LIN {X 0,Y 418.203,Z 303.395,A -85,B 0,C 180,E1 -10039.132,E2 -10039.132} C_VEL
LIN {X 0,Y 418.231,Z 303.386,A -85,B 0,C 180,E1 -10042.775,E2 -10042.775} C_VEL
LIN {X 0,Y 418.224,Z 303.373,A -85,B 0,C 180,E1 -10046.321,E2 -10046.321} C_VEL
LIN {X 0,Y 418.233,Z 303.387,A -85,B 0,C 180,E1 -10049.727,E2 -10049.727} C_VEL
LIN {X 0,Y 418.217,Z 303.388,A -85,B 0,C 180,E1 -10053.017,E2 -10053.017} C_VEL
LIN {X 0,Y 418.247,Z 303.384,A -85,B 0,C 180,E1 -10056.217,E2 -10056.217} C_VEL
LIN {X 0,Y 418.24,Z 303.384,A -85,B 0,C 180,E1 -10059.337,E2 -10059.337} C_VEL
LIN {X 0,Y 418.246,Z 303.382,A -85,B 0,C 180,E1 -10062.395,E2 -10062.395} C_VEL
LIN {X 0,Y 418.265,Z 303.381,A -85,B 0,C 180,E1 -10065.402,E2 -10065.402} C_VEL
LIN {X 0,Y 418.292,Z 303.381,A -85,B 0,C 180,E1 -10068.369,E2 -10068.369} C_VEL
LIN {X 0,Y 418.437,Z 303.357,A -85,B 0,C 180,E1 -10072.278,E2 -10072.278} C_VEL
LIN {X 0,Y 418.453,Z 303.363,A -85,B 0,C 180,E1 -10074.217,E2 -10074.217} C_VEL
LIN {X 0,Y 418.521,Z 303.346,A -85,B 0,C 180,E1 -10078.076,E2 -10078.076} C_VEL
LIN {X 0,Y 418.461,Z 303.353,A -85,B 0,C 180,E1 -10080.963,E2 -10080.963} C_VEL
LIN {X 0,Y 418.457,Z 303.356,A -85,B 0,C 180,E1 -10082.888,E2 -10082.888} C_VEL
LIN {X 0,Y 418.488,Z 303.352,A -85,B 0,C 180,E1 -10085.783,E2 -10085.783} C_VEL
LIN {X 0,Y 418.36,Z 303.365,A -85,B 0,C 180,E1 -10088.696,E2 -10088.696} C_VEL
LIN {X 0,Y 418.302,Z 303.372,A -85,B 0,C 180,E1 -10091.632,E2 -10091.632} C_VEL
LIN {X 0,Y 418.289,Z 303.374,A -85,B 0,C 180,E1 -10094.598,E2 -10094.598} C_VEL
LIN {X 0,Y 418.27,Z 303.372,A -85,B 0,C 180,E1 -10097.605,E2 -10097.605} C_VEL
LIN {X 0,Y 418.242,Z 303.384,A -85,B 0,C 180,E1 -10100.664,E2 -10100.664} C_VEL
LIN {X 0,Y 418.251,Z 303.38,A -85,B 0,C 180,E1 -10103.784,E2 -10103.784} C_VEL
LIN {X 0,Y 418.217,Z 303.387,A -85,B 0,C 180,E1 -10107.048,E2 -10107.048} C_VEL
LIN {X 0,Y 418.235,Z 303.384,A -85,B 0,C 180,E1 -10110.273,E2 -10110.273} C_VEL
LIN {X 0,Y 418.242,Z 303.388,A -85,B 0,C 180,E1 -10113.678,E2 -10113.678} C_VEL
LIN {X 0,Y 418.232,Z 303.388,A -85,B 0,C 180,E1 -10117.225,E2 -10117.225} C_VEL
LIN {X 0,Y 418.207,Z 303.39,A -85,B 0,C 180,E1 -10120.869,E2 -10120.869} C_VEL
LIN {X 0,Y 418.203,Z 303.38,A -85,B 0,C 180,E1 -10123.73,E2 -10123.73} C_VEL
LIN {X 0,Y 418.203,Z 303.392,A -85,B 0,C 180,E1 -10126.449,E2 -10126.449} C_VEL
LIN {X 0,Y 418.217,Z 303.391,A -85,B 0,C 180,E1 -10129.132,E2 -10129.132} C_VEL
LIN {X 0,Y 418.221,Z 303.393,A -85,B 0,C 180,E1 -10132.168,E2 -10132.168} C_VEL
LIN {X 0,Y 418.262,Z 303.379,A -85,B 0,C 180,E1 -10135.421,E2 -10135.421} C_VEL
LIN {X 0,Y 418.21,Z 303.393,A -85,B 0,C 180,E1 -10138.605,E2 -10138.605} C_VEL
LIN {X 0,Y 418.318,Z 303.393,A -85,B 0,C 180,E1 -10142.251,E2 -10142.251} C_VEL
LIN {X 0,Y 420.764,Z 315.163,A -85,B 0,C 180,E1 -10144.934,E2 -10144.934} C_VEL
LIN {X 0,Y 421.568,Z 320.765,A -85,B 0,C 180,E1 -10146.155,E2 -10146.155} C_VEL
LIN {X 0,Y 420.324,Z 337.886,A -85,B 0,C 180,E1 -10149.597,E2 -10149.597} C_VEL
LIN {X 0,Y 420,Z 342.885,A -85,B 0,C 180,E1 -10150.591,E2 -10150.591} C_VEL
LIN {X 0,Y 423.729,Z 363.444,A -85,B 0,C 180,E1 -10151.164,E2 -10151.164} C_VEL
LIN {X 0,Y 424.474,Z 370.034,A -85,B 0,C 180,E1 -10151.321,E2 -10151.321} C_VEL
LIN {X 0,Y 423.504,Z 451.222,A -85,B 0,C 180,E1 -10152.746,E2 -10152.746} C_VEL
LIN {X 0,Y 422.93,Z 464.392,A -85,B 0,C 180,E1 -10153.157,E2 -10153.157} C_VEL
LIN {X 0,Y 422.257,Z 477.049,A -85,B 0,C 180,E1 -10153.751,E2 -10153.751} C_VEL
LIN {X 0,Y 421.448,Z 489.124,A -85,B 0,C 180,E1 -10154.526,E2 -10154.526} C_VEL
LIN {X 0,Y 420.581,Z 500.615,A -85,B 0,C 180,E1 -10155.485,E2 -10155.485} C_VEL
LIN {X 0,Y 419.836,Z 510.983,A -85,B 0,C 180,E1 -10156.571,E2 -10156.571} C_VEL
LIN {X 0,Y 419.198,Z 519.483,A -85,B 0,C 180,E1 -10157.658,E2 -10157.658} C_VEL
LIN {X 0,Y 418.464,Z 527.341,A -85,B 0,C 180,E1 -10158.865,E2 -10158.865} C_VEL
LIN {X 0,Y 417.91,Z 535.031,A -85,B 0,C 180,E1 -10160.32,E2 -10160.32} C_VEL
LIN {X 0,Y 417.502,Z 541.222,A -85,B 0,C 180,E1 -10161.775,E2 -10161.775} C_VEL
LIN {X 0,Y 417.242,Z 546.152,A -85,B 0,C 180,E1 -10163.23,E2 -10163.23} C_VEL
LIN {X 0,Y 417.122,Z 549.965,A -85,B 0,C 180,E1 -10164.684,E2 -10164.684} C_VEL
LIN {X 0,Y 417.013,Z 552.763,A -85,B 0,C 180,E1 -10166.136,E2 -10166.136} C_VEL
LIN {X 0,Y 417.056,Z 555.025,A -85,B 0,C 180,E1 -10168.069,E2 -10168.069} C_VEL
LIN {X 0,Y 417.011,Z 555.562,A -85,B 0,C 180,E1 -10169.035,E2 -10169.035} C_VEL
LIN {X 0,Y 417.004,Z 555.667,A -85,B 0,C 180,E1 -10170.001,E2 -10170.001} C_VEL
LIN {X 0,Y 417.056,Z 554.713,A -85,B 0,C 180,E1 -10171.932,E2 -10171.932} C_VEL
LIN {X 0,Y 417.03,Z 553.643,A -85,B 0,C 180,E1 -10172.899,E2 -10172.899} C_VEL
LIN {X 0,Y 417.015,Z 552.117,A -85,B 0,C 180,E1 -10173.866,E2 -10173.866} C_VEL
LIN {X 0,Y 417.122,Z 549.039,A -85,B 0,C 180,E1 -10175.318,E2 -10175.318} C_VEL
LIN {X 0,Y 417.233,Z 544.889,A -85,B 0,C 180,E1 -10176.772,E2 -10176.772} C_VEL
LIN {X 0,Y 417.504,Z 538.537,A -85,B 0,C 180,E1 -10178.471,E2 -10178.471} C_VEL
LIN {X 0,Y 417.901,Z 531.613,A -85,B 0,C 180,E1 -10179.927,E2 -10179.927} C_VEL
LIN {X 0,Y 418.308,Z 524.531,A -85,B 0,C 180,E1 -10181.141,E2 -10181.141} C_VEL
LIN {X 0,Y 418.943,Z 515.991,A -85,B 0,C 180,E1 -10182.351,E2 -10182.351} C_VEL
LIN {X 0,Y 419.634,Z 505.417,A -85,B 0,C 180,E1 -10183.561,E2 -10183.561} C_VEL
LIN {X 0,Y 420.269,Z 494.939,A -85,B 0,C 180,E1 -10184.528,E2 -10184.528} C_VEL
LIN {X 0,Y 420.952,Z 483.424,A -85,B 0,C 180,E1 -10185.37,E2 -10185.37} C_VEL
LIN {X 0,Y 421.546,Z 471.495,A -85,B 0,C 180,E1 -10186.03,E2 -10186.03} C_VEL
LIN {X 0,Y 422.09,Z 458.63,A -85,B 0,C 180,E1 -10186.537,E2 -10186.537} C_VEL
LIN {X 0,Y 422.434,Z 445.189,A -85,B 0,C 180,E1 -10186.865,E2 -10186.865} C_VEL
LIN {X 0,Y 423.121,Z 367.493,A -85,B 0,C 180,E1 -10188.19,E2 -10188.19} C_VEL
LIN {X 0,Y 419.458,Z 343.088,A -85,B 0,C 180,E1 -10188.785,E2 -10188.785} C_VEL
LIN {X 0,Y 420.548,Z 324.975,A -85,B 0,C 180,E1 -10192.346,E2 -10192.346} C_VEL
LIN {X 0,Y 420.862,Z 317.24,A -85,B 0,C 180,E1 -10193.889,E2 -10193.889} C_VEL
LIN {X 0,Y 418.323,Z 303.378,A -85,B 0,C 180,E1 -10196.875,E2 -10196.875} C_VEL
LIN {X 0,Y 418.249,Z 303.384,A -85,B 0,C 180,E1 -10200.272,E2 -10200.272} C_VEL
LIN {X 0,Y 418.253,Z 303.385,A -85,B 0,C 180,E1 -10203.677,E2 -10203.677} C_VEL
LIN {X 0,Y 418.242,Z 303.382,A -85,B 0,C 180,E1 -10207.225,E2 -10207.225} C_VEL
LIN {X 0,Y 418.213,Z 303.387,A -85,B 0,C 180,E1 -10210.868,E2 -10210.868} C_VEL
LIN {X 0,Y 418.212,Z 303.387,A -85,B 0,C 180,E1 -10213.729,E2 -10213.729} C_VEL
LIN {X 0,Y 418.212,Z 303.394,A -85,B 0,C 180,E1 -10216.449,E2 -10216.449} C_VEL
LIN {X 0,Y 418.225,Z 303.385,A -85,B 0,C 180,E1 -10219.131,E2 -10219.131} C_VEL
LIN {X 0,Y 418.228,Z 303.386,A -85,B 0,C 180,E1 -10222.168,E2 -10222.168} C_VEL
LIN {X 0,Y 418.269,Z 303.38,A -85,B 0,C 180,E1 -10225.42,E2 -10225.42} C_VEL
LIN {X 0,Y 418.215,Z 303.389,A -85,B 0,C 180,E1 -10228.604,E2 -10228.604} C_VEL
LIN {X 0,Y 418.265,Z 303.379,A -85,B 0,C 180,E1 -10231.934,E2 -10231.934} C_VEL
LIN {X 0,Y 418.276,Z 303.386,A -85,B 0,C 180,E1 -10235.162,E2 -10235.162} C_VEL
LIN {X 0,Y 418.238,Z 303.382,A -85,B 0,C 180,E1 -10238.304,E2 -10238.304} C_VEL
LIN {X 0,Y 418.281,Z 303.385,A -85,B 0,C 180,E1 -10241.383,E2 -10241.383} C_VEL
LIN {X 0,Y 418.305,Z 303.374,A -85,B 0,C 180,E1 -10244.406,E2 -10244.406} C_VEL
LIN {X 0,Y 418.359,Z 303.372,A -85,B 0,C 180,E1 -10247.385,E2 -10247.385} C_VEL
LIN {X 0,Y 418.34,Z 303.371,A -85,B 0,C 180,E1 -10250.328,E2 -10250.328} C_VEL
LIN {X 0,Y 418.471,Z 303.355,A -85,B 0,C 180,E1 -10253.248,E2 -10253.248} C_VEL
LIN {X 0,Y 418.331,Z 303.371,A -85,B 0,C 180,E1 -10255.181,E2 -10255.181} C_VEL
LIN {X 0,Y 418.542,Z 303.352,A -85,B 0,C 180,E1 -10258.075,E2 -10258.075} C_VEL
LIN {X 0,Y 418.67,Z 303.335,A -85,B 0,C 180,E1 -10260,E2 -10260} C_VEL
LIN {X 0,Y 418.494,Z 303.351,A -85,B 0,C 180,E1 -10262.888,E2 -10262.888} C_VEL
LIN {X 0,Y 418.447,Z 303.358,A -85,B 0,C 180,E1 -10266.548,E2 -10266.548} C_VEL
LIN {X 0,Y 418.342,Z 303.37,A -85,B 0,C 180,E1 -10269.671,E2 -10269.671} C_VEL
LIN {X 0,Y 418.35,Z 303.372,A -85,B 0,C 180,E1 -10273,E2 -10273} C_VEL
LIN {X 0,Y 418.316,Z 303.381,A -85,B 0,C 180,E1 -10276.735,E2 -10276.735} C_VEL
LIN {X 0,Y 418.273,Z 303.378,A -85,B 0,C 180,E1 -10279.79,E2 -10279.79} C_VEL
LIN {X 0,Y 418.234,Z 303.388,A -85,B 0,C 180,E1 -10282.736,E2 -10282.736} C_VEL
LIN {X 0,Y 418.24,Z 303.383,A -85,B 0,C 180,E1 -10285.906,E2 -10285.906} C_VEL
LIN {X 0,Y 418.263,Z 303.387,A -85,B 0,C 180,E1 -10289.162,E2 -10289.162} C_VEL
LIN {X 0,Y 418.259,Z 303.382,A -85,B 0,C 180,E1 -10292.843,E2 -10292.843} C_VEL
LIN {X 0,Y 418.245,Z 303.382,A -85,B 0,C 180,E1 -10296.237,E2 -10296.237} C_VEL
LIN {X 0,Y 418.244,Z 303.389,A -85,B 0,C 180,E1 -10299.683,E2 -10299.683} C_VEL
LIN {X 0,Y 418.225,Z 303.385,A -85,B 0,C 180,E1 -10302.32,E2 -10302.32} C_VEL
LIN {X 0,Y 418.237,Z 303.383,A -85,B 0,C 180,E1 -10305.108,E2 -10305.108} C_VEL
LIN {X 0,Y 418.236,Z 303.389,A -85,B 0,C 180,E1 -10307.765,E2 -10307.765} C_VEL
LIN {X 0,Y 418.244,Z 303.384,A -85,B 0,C 180,E1 -10311.556,E2 -10311.556} C_VEL
LIN {X 0,Y 418.26,Z 303.38,A -85,B 0,C 180,E1 -10315.158,E2 -10315.158} C_VEL
LIN {X 0,Y 418.247,Z 303.381,A -85,B 0,C 180,E1 -10317.471,E2 -10317.471} C_VEL
LIN {X 0,Y 418.266,Z 303.382,A -85,B 0,C 180,E1 -10320.896,E2 -10320.896} C_VEL
LIN {X 0,Y 418.238,Z 303.385,A -85,B 0,C 180,E1 -10324.093,E2 -10324.093} C_VEL
LIN {X 0,Y 418.238,Z 303.384,A -85,B 0,C 180,E1 -10327.263,E2 -10327.263} C_VEL
LIN {X 0,Y 418.284,Z 303.379,A -85,B 0,C 180,E1 -10330.363,E2 -10330.363} C_VEL
LIN {X 0,Y 418.317,Z 303.375,A -85,B 0,C 180,E1 -10333.404,E2 -10333.404} C_VEL
LIN {X 0,Y 418.347,Z 303.376,A -85,B 0,C 180,E1 -10336.999,E2 -10336.999} C_VEL
LIN {X 0,Y 418.357,Z 303.373,A -85,B 0,C 180,E1 -10340.816,E2 -10340.816} C_VEL
LIN {X 0,Y 418.382,Z 303.531,A -85,B 0,C 180,E1 -10341.304,E2 -10341.304} C_VEL
LIN {X 0,Y 419.874,Z 311.987,A -85,B 0,C 180,E1 -10343.27,E2 -10343.27} C_VEL
LIN {X 0,Y 419.639,Z 321.318,A -85,B 0,C 180,E1 -10345.314,E2 -10345.314} C_VEL
LIN {X 0,Y 423.403,Z 342.206,A -85,B 0,C 180,E1 -10345.831,E2 -10345.831} C_VEL
LIN {X 0,Y 422.409,Z 428.625,A -85,B 0,C 180,E1 -10347.32,E2 -10347.32} C_VEL
LIN {X 0,Y 422.171,Z 435.313,A -85,B 0,C 180,E1 -10347.505,E2 -10347.505} C_VEL
LIN {X 0,Y 420.767,Z 442.88,A -85,B 0,C 180,E1 -10347.736,E2 -10347.736} C_VEL
LIN {X 0,Y 418.093,Z 450.166,A -85,B 0,C 180,E1 -10347.981,E2 -10347.981} C_VEL
LIN {X 0,Y 415.016,Z 459.136,A -85,B 0,C 180,E1 -10348.398,E2 -10348.398} C_VEL
LIN {X 0,Y 414.153,Z 464.405,A -85,B 0,C 180,E1 -10348.731,E2 -10348.731} C_VEL
LIN {X 0,Y 413.477,Z 475.677,A -85,B 0,C 180,E1 -10349.634,E2 -10349.634} C_VEL
LIN {X 0,Y 412.722,Z 486.46,A -85,B 0,C 180,E1 -10350.731,E2 -10350.731} C_VEL
LIN {X 0,Y 412.056,Z 496.153,A -85,B 0,C 180,E1 -10351.954,E2 -10351.954} C_VEL
LIN {X 0,Y 411.442,Z 504.117,A -85,B 0,C 180,E1 -10353.181,E2 -10353.181} C_VEL
LIN {X 0,Y 410.924,Z 511.91,A -85,B 0,C 180,E1 -10354.659,E2 -10354.659} C_VEL
LIN {X 0,Y 410.603,Z 518.384,A -85,B 0,C 180,E1 -10356.208,E2 -10356.208} C_VEL
LIN {X 0,Y 410.256,Z 523.824,A -85,B 0,C 180,E1 -10357.876,E2 -10357.876} C_VEL
LIN {X 0,Y 410.051,Z 527.487,A -85,B 0,C 180,E1 -10359.37,E2 -10359.37} C_VEL
LIN {X 0,Y 409.963,Z 530.119,A -85,B 0,C 180,E1 -10360.869,E2 -10360.869} C_VEL
LIN {X 0,Y 409.905,Z 531.676,A -85,B 0,C 180,E1 -10362.235,E2 -10362.235} C_VEL
LIN {X 0,Y 409.789,Z 532.527,A -85,B 0,C 180,E1 -10363.892,E2 -10363.892} C_VEL
LIN {X 0,Y 409.806,Z 532.503,A -85,B 0,C 180,E1 -10364.906,E2 -10364.906} C_VEL
LIN {X 0,Y 409.886,Z 531.827,A -85,B 0,C 180,E1 -10366.222,E2 -10366.222} C_VEL
LIN {X 0,Y 409.974,Z 529.837,A -85,B 0,C 180,E1 -10367.972,E2 -10367.972} C_VEL
LIN {X 0,Y 410.241,Z 526.867,A -85,B 0,C 180,E1 -10369.572,E2 -10369.572} C_VEL
LIN {X 0,Y 410.504,Z 523.013,A -85,B 0,C 180,E1 -10371.07,E2 -10371.07} C_VEL
LIN {X 0,Y 410.967,Z 517.198,A -85,B 0,C 180,E1 -10372.785,E2 -10372.785} C_VEL
LIN {X 0,Y 411.614,Z 509.788,A -85,B 0,C 180,E1 -10374.458,E2 -10374.458} C_VEL
LIN {X 0,Y 412.182,Z 502.894,A -85,B 0,C 180,E1 -10375.717,E2 -10375.717} C_VEL
LIN {X 0,Y 412.992,Z 493.798,A -85,B 0,C 180,E1 -10377.077,E2 -10377.077} C_VEL
LIN {X 0,Y 413.829,Z 484.223,A -85,B 0,C 180,E1 -10378.232,E2 -10378.232} C_VEL
LIN {X 0,Y 414.719,Z 473.231,A -85,B 0,C 180,E1 -10379.295,E2 -10379.295} C_VEL
LIN {X 0,Y 415.533,Z 461.267,A -85,B 0,C 180,E1 -10380.209,E2 -10380.209} C_VEL
LIN {X 0,Y 416.24,Z 448.697,A -85,B 0,C 180,E1 -10380.924,E2 -10380.924} C_VEL
LIN {X 0,Y 416.732,Z 435.712,A -85,B 0,C 180,E1 -10381.448,E2 -10381.448} C_VEL
LIN {X 0,Y 417.033,Z 422.429,A -85,B 0,C 180,E1 -10381.777,E2 -10381.777} C_VEL
LIN {X 0,Y 418.216,Z 343.018,A -85,B 0,C 180,E1 -10383.163,E2 -10383.163} C_VEL
LIN {X 0,Y 413.927,Z 323.175,A -85,B 0,C 180,E1 -10383.775,E2 -10383.775} C_VEL
LIN {X 0,Y 413.523,Z 321.336,A -85,B 0,C 180,E1 -10383.87,E2 -10383.87} C_VEL
LIN {X 0,Y 413.629,Z 316.261,A -85,B 0,C 180,E1 -10384.99,E2 -10384.99} C_VEL
LIN {X 0,Y 411.392,Z 305.21,A -85,B 0,C 180,E1 -10387.641,E2 -10387.641} C_VEL
LIN {X 0,Y 411.195,Z 304.267,A -85,B 0,C 180,E1 -10387.894,E2 -10387.894} C_VEL
LIN {X 0,Y 411.145,Z 304.269,A -85,B 0,C 180,E1 -10391.226,E2 -10391.226} C_VEL
LIN {X 0,Y 411.168,Z 304.269,A -85,B 0,C 180,E1 -10394.49,E2 -10394.49} C_VEL
LIN {X 0,Y 411.156,Z 304.266,A -85,B 0,C 180,E1 -10398.192,E2 -10398.192} C_VEL
LIN {X 0,Y 411.188,Z 304.263,A -85,B 0,C 180,E1 -10401.832,E2 -10401.832} C_VEL
LIN {X 0,Y 411.195,Z 304.258,A -85,B 0,C 180,E1 -10405.123,E2 -10405.123} C_VEL
LIN {X 0,Y 411.155,Z 304.269,A -85,B 0,C 180,E1 -10408.002,E2 -10408.002} C_VEL
LIN {X 0,Y 411.184,Z 304.264,A -85,B 0,C 180,E1 -10411.408,E2 -10411.408} C_VEL
LIN {X 0,Y 411.203,Z 304.258,A -85,B 0,C 180,E1 -10414.934,E2 -10414.934} C_VEL
LIN {X 0,Y 411.194,Z 304.261,A -85,B 0,C 180,E1 -10417.913,E2 -10417.913} C_VEL
LIN {X 0,Y 411.205,Z 304.259,A -85,B 0,C 180,E1 -10421.051,E2 -10421.051} C_VEL
LIN {X 0,Y 411.199,Z 304.265,A -85,B 0,C 180,E1 -10424.13,E2 -10424.13} C_VEL
LIN {X 0,Y 411.292,Z 304.242,A -85,B 0,C 180,E1 -10427.166,E2 -10427.166} C_VEL
LIN {X 0,Y 411.264,Z 304.253,A -85,B 0,C 180,E1 -10430.161,E2 -10430.161} C_VEL
LIN {X 0,Y 411.375,Z 304.237,A -85,B 0,C 180,E1 -10433.132,E2 -10433.132} C_VEL
LIN {X 0,Y 411.271,Z 304.249,A -85,B 0,C 180,E1 -10435.099,E2 -10435.099} C_VEL
LIN {X 0,Y 411.49,Z 304.222,A -85,B 0,C 180,E1 -10438.043,E2 -10438.043} C_VEL
LIN {X 0,Y 411.426,Z 304.229,A -85,B 0,C 180,E1 -10440.979,E2 -10440.979} C_VEL
LIN {X 0,Y 411.415,Z 304.233,A -85,B 0,C 180,E1 -10442.938,E2 -10442.938} C_VEL
LIN {X 0,Y 411.422,Z 304.228,A -85,B 0,C 180,E1 -10446.868,E2 -10446.868} C_VEL
LIN {X 0,Y 411.273,Z 304.249,A -85,B 0,C 180,E1 -10449.839,E2 -10449.839} C_VEL
LIN {X 0,Y 411.297,Z 304.243,A -85,B 0,C 180,E1 -10453.104,E2 -10453.104} C_VEL
LIN {X 0,Y 411.249,Z 304.255,A -85,B 0,C 180,E1 -10456.889,E2 -10456.889} C_VEL
LIN {X 0,Y 411.223,Z 304.255,A -85,B 0,C 180,E1 -10459.987,E2 -10459.987} C_VEL
LIN {X 0,Y 411.181,Z 304.26,A -85,B 0,C 180,E1 -10463.149,E2 -10463.149} C_VEL
LIN {X 0,Y 411.177,Z 304.262,A -85,B 0,C 180,E1 -10466.385,E2 -10466.385} C_VEL
LIN {X 0,Y 411.191,Z 304.265,A -85,B 0,C 180,E1 -10469.714,E2 -10469.714} C_VEL
LIN {X 0,Y 411.2,Z 304.263,A -85,B 0,C 180,E1 -10473.157,E2 -10473.157} C_VEL
LIN {X 0,Y 411.186,Z 304.262,A -85,B 0,C 180,E1 -10476.553,E2 -10476.553} C_VEL
LIN {X 0,Y 411.171,Z 304.268,A -85,B 0,C 180,E1 -10479.723,E2 -10479.723} C_VEL
LIN {X 0,Y 411.165,Z 304.256,A -85,B 0,C 180,E1 -10483.135,E2 -10483.135} C_VEL
LIN {X 0,Y 411.163,Z 304.274,A -85,B 0,C 180,E1 -10485.882,E2 -10485.882} C_VEL
LIN {X 0,Y 411.156,Z 304.27,A -85,B 0,C 180,E1 -10488.773,E2 -10488.773} C_VEL
LIN {X 0,Y 411.186,Z 304.269,A -85,B 0,C 180,E1 -10492.027,E2 -10492.027} C_VEL
LIN {X 0,Y 411.203,Z 304.259,A -85,B 0,C 180,E1 -10495.668,E2 -10495.668} C_VEL
LIN {X 0,Y 411.187,Z 304.267,A -85,B 0,C 180,E1 -10499.154,E2 -10499.154} C_VEL
LIN {X 0,Y 411.265,Z 304.258,A -85,B 0,C 180,E1 -10501.902,E2 -10501.902} C_VEL
LIN {X 0,Y 413.59,Z 315.249,A -85,B 0,C 180,E1 -10504.471,E2 -10504.471} C_VEL
LIN {X 0,Y 414.671,Z 322.091,A -85,B 0,C 180,E1 -10506,E2 -10506} C_VEL
LIN {X 0,Y 413.41,Z 338.62,A -85,B 0,C 180,E1 -10509.38,E2 -10509.38} C_VEL
LIN {X 0,Y 413.181,Z 342.913,A -85,B 0,C 180,E1 -10510.208,E2 -10510.208} C_VEL
LIN {X 0,Y 417.065,Z 363.859,A -85,B 0,C 180,E1 -10510.814,E2 -10510.814} C_VEL
LIN {X 0,Y 417.867,Z 370.718,A -85,B 0,C 180,E1 -10510.983,E2 -10510.983} C_VEL
LIN {X 0,Y 416.829,Z 451.568,A -85,B 0,C 180,E1 -10512.429,E2 -10512.429} C_VEL
LIN {X 0,Y 416.203,Z 464.561,A -85,B 0,C 180,E1 -10512.845,E2 -10512.845} C_VEL
LIN {X 0,Y 415.484,Z 477.666,A -85,B 0,C 180,E1 -10513.479,E2 -10513.479} C_VEL
LIN {X 0,Y 414.636,Z 489.507,A -85,B 0,C 180,E1 -10514.266,E2 -10514.266} C_VEL
LIN {X 0,Y 413.735,Z 500.891,A -85,B 0,C 180,E1 -10515.239,E2 -10515.239} C_VEL
LIN {X 0,Y 412.922,Z 511.174,A -85,B 0,C 180,E1 -10516.341,E2 -10516.341} C_VEL
LIN {X 0,Y 412.25,Z 519.598,A -85,B 0,C 180,E1 -10517.447,E2 -10517.447} C_VEL
LIN {X 0,Y 411.368,Z 528.752,A -85,B 0,C 180,E1 -10518.92,E2 -10518.92} C_VEL
LIN {X 0,Y 410.8,Z 536.134,A -85,B 0,C 180,E1 -10520.399,E2 -10520.399} C_VEL
LIN {X 0,Y 410.345,Z 542.951,A -85,B 0,C 180,E1 -10522.126,E2 -10522.126} C_VEL
LIN {X 0,Y 410.043,Z 547.898,A -85,B 0,C 180,E1 -10523.776,E2 -10523.776} C_VEL
LIN {X 0,Y 410.019,Z 550.906,A -85,B 0,C 180,E1 -10525.084,E2 -10525.084} C_VEL
LIN {X 0,Y 409.924,Z 553.935,A -85,B 0,C 180,E1 -10527.053,E2 -10527.053} C_VEL
LIN {X 0,Y 409.966,Z 554.858,A -85,B 0,C 180,E1 -10528.036,E2 -10528.036} C_VEL
LIN {X 0,Y 409.935,Z 555.373,A -85,B 0,C 180,E1 -10529.019,E2 -10529.019} C_VEL
LIN {X 0,Y 409.936,Z 555.165,A -85,B 0,C 180,E1 -10530.983,E2 -10530.983} C_VEL
LIN {X 0,Y 409.967,Z 554.482,A -85,B 0,C 180,E1 -10531.966,E2 -10531.966} C_VEL
LIN {X 0,Y 409.929,Z 553.39,A -85,B 0,C 180,E1 -10532.949,E2 -10532.949} C_VEL
LIN {X 0,Y 409.933,Z 551.846,A -85,B 0,C 180,E1 -10533.933,E2 -10533.933} C_VEL
LIN {X 0,Y 410.018,Z 548.738,A -85,B 0,C 180,E1 -10535.41,E2 -10535.41} C_VEL
LIN {X 0,Y 410.166,Z 544.559,A -85,B 0,C 180,E1 -10536.89,E2 -10536.89} C_VEL
LIN {X 0,Y 410.465,Z 538.174,A -85,B 0,C 180,E1 -10538.617,E2 -10538.617} C_VEL
LIN {X 0,Y 410.869,Z 531.21,A -85,B 0,C 180,E1 -10540.099,E2 -10540.099} C_VEL
LIN {X 0,Y 411.447,Z 522.469,A -85,B 0,C 180,E1 -10541.579,E2 -10541.579} C_VEL
LIN {X 0,Y 412.041,Z 513.502,A -85,B 0,C 180,E1 -10542.812,E2 -10542.812} C_VEL
LIN {X 0,Y 412.738,Z 503.516,A -85,B 0,C 180,E1 -10543.931,E2 -10543.931} C_VEL
LIN {X 0,Y 413.441,Z 492.77,A -85,B 0,C 180,E1 -10544.899,E2 -10544.899} C_VEL
LIN {X 0,Y 414.181,Z 480.553,A -85,B 0,C 180,E1 -10545.754,E2 -10545.754} C_VEL
LIN {X 0,Y 414.787,Z 467.759,A -85,B 0,C 180,E1 -10546.425,E2 -10546.425} C_VEL
LIN {X 0,Y 415.299,Z 455.049,A -85,B 0,C 180,E1 -10546.879,E2 -10546.879} C_VEL
LIN {X 0,Y 415.651,Z 437.061,A -85,B 0,C 180,E1 -10547.244,E2 -10547.244} C_VEL
LIN {X 0,Y 416.352,Z 369.112,A -85,B 0,C 180,E1 -10548.418,E2 -10548.418} C_VEL
LIN {X 0,Y 412.506,Z 342.976,A -85,B 0,C 180,E1 -10549.049,E2 -10549.049} C_VEL
LIN {X 0,Y 413.653,Z 324.528,A -85,B 0,C 180,E1 -10552.739,E2 -10552.739} C_VEL
LIN {X 0,Y 413.859,Z 318.067,A -85,B 0,C 180,E1 -10554.052,E2 -10554.052} C_VEL
LIN {X 0,Y 411.288,Z 304.255,A -85,B 0,C 180,E1 -10557.096,E2 -10557.096} C_VEL
LIN {X 0,Y 411.205,Z 304.266,A -85,B 0,C 180,E1 -10559.713,E2 -10559.713} C_VEL
LIN {X 0,Y 411.211,Z 304.258,A -85,B 0,C 180,E1 -10563.156,E2 -10563.156} C_VEL
LIN {X 0,Y 411.196,Z 304.262,A -85,B 0,C 180,E1 -10566.553,E2 -10566.553} C_VEL
LIN {X 0,Y 411.174,Z 304.265,A -85,B 0,C 180,E1 -10569.721,E2 -10569.721} C_VEL
LIN {X 0,Y 411.174,Z 304.263,A -85,B 0,C 180,E1 -10573.134,E2 -10573.134} C_VEL
LIN {X 0,Y 411.172,Z 304.264,A -85,B 0,C 180,E1 -10575.881,E2 -10575.881} C_VEL
LIN {X 0,Y 411.165,Z 304.268,A -85,B 0,C 180,E1 -10578.772,E2 -10578.772} C_VEL
LIN {X 0,Y 411.193,Z 304.261,A -85,B 0,C 180,E1 -10582.026,E2 -10582.026} C_VEL
LIN {X 0,Y 411.21,Z 304.258,A -85,B 0,C 180,E1 -10585.667,E2 -10585.667} C_VEL
LIN {X 0,Y 411.193,Z 304.265,A -85,B 0,C 180,E1 -10589.152,E2 -10589.152} C_VEL
LIN {X 0,Y 411.212,Z 304.259,A -85,B 0,C 180,E1 -10592.519,E2 -10592.519} C_VEL
LIN {X 0,Y 411.215,Z 304.259,A -85,B 0,C 180,E1 -10595.784,E2 -10595.784} C_VEL
LIN {X 0,Y 411.201,Z 304.263,A -85,B 0,C 180,E1 -10598.966,E2 -10598.966} C_VEL
LIN {X 0,Y 411.25,Z 304.254,A -85,B 0,C 180,E1 -10602.085,E2 -10602.085} C_VEL
LIN {X 0,Y 411.263,Z 304.254,A -85,B 0,C 180,E1 -10605.147,E2 -10605.147} C_VEL
LIN {X 0,Y 411.286,Z 304.25,A -85,B 0,C 180,E1 -10608.167,E2 -10608.167} C_VEL
LIN {X 0,Y 411.442,Z 304.232,A -85,B 0,C 180,E1 -10612.192,E2 -10612.192} C_VEL
LIN {X 0,Y 411.466,Z 304.231,A -85,B 0,C 180,E1 -10614.118,E2 -10614.118} C_VEL
LIN {X 0,Y 411.511,Z 304.229,A -85,B 0,C 180,E1 -10618.042,E2 -10618.042} C_VEL
LIN {X 0,Y 411.639,Z 304.211,A -85,B 0,C 180,E1 -10620,E2 -10620} C_VEL
LIN {X 0,Y 411.451,Z 304.229,A -85,B 0,C 180,E1 -10622.937,E2 -10622.937} C_VEL
LIN {X 0,Y 411.396,Z 304.235,A -85,B 0,C 180,E1 -10626.545,E2 -10626.545} C_VEL
LIN {X 0,Y 411.322,Z 304.247,A -85,B 0,C 180,E1 -10628.846,E2 -10628.846} C_VEL
LIN {X 0,Y 411.286,Z 304.249,A -85,B 0,C 180,E1 -10631.832,E2 -10631.832} C_VEL
LIN {X 0,Y 411.264,Z 304.257,A -85,B 0,C 180,E1 -10634.852,E2 -10634.852} C_VEL
LIN {X 0,Y 411.249,Z 304.253,A -85,B 0,C 180,E1 -10637.915,E2 -10637.915} C_VEL
LIN {X 0,Y 411.199,Z 304.266,A -85,B 0,C 180,E1 -10641.034,E2 -10641.034} C_VEL
LIN {X 0,Y 411.214,Z 304.258,A -85,B 0,C 180,E1 -10644.216,E2 -10644.216} C_VEL
LIN {X 0,Y 411.21,Z 304.262,A -85,B 0,C 180,E1 -10647.481,E2 -10647.481} C_VEL
LIN {X 0,Y 411.191,Z 304.263,A -85,B 0,C 180,E1 -10650.847,E2 -10650.847} C_VEL
LIN {X 0,Y 411.206,Z 304.258,A -85,B 0,C 180,E1 -10654.333,E2 -10654.333} C_VEL
LIN {X 0,Y 411.191,Z 304.263,A -85,B 0,C 180,E1 -10657.974,E2 -10657.974} C_VEL
LIN {X 0,Y 411.162,Z 304.266,A -85,B 0,C 180,E1 -10661.227,E2 -10661.227} C_VEL
LIN {X 0,Y 411.178,Z 304.263,A -85,B 0,C 180,E1 -10664.49,E2 -10664.49} C_VEL
LIN {X 0,Y 411.174,Z 304.267,A -85,B 0,C 180,E1 -10668.193,E2 -10668.193} C_VEL
LIN {X 0,Y 411.204,Z 304.259,A -85,B 0,C 180,E1 -10670.774,E2 -10670.774} C_VEL
LIN {X 0,Y 411.199,Z 304.264,A -85,B 0,C 180,E1 -10674.471,E2 -10674.471} C_VEL
LIN {X 0,Y 411.209,Z 304.26,A -85,B 0,C 180,E1 -10676.873,E2 -10676.873} C_VEL
LIN {X 0,Y 411.214,Z 304.263,A -85,B 0,C 180,E1 -10680.649,E2 -10680.649} C_VEL
LIN {X 0,Y 411.204,Z 304.259,A -85,B 0,C 180,E1 -10683.616,E2 -10683.616} C_VEL
LIN {X 0,Y 411.203,Z 304.265,A -85,B 0,C 180,E1 -10686.852,E2 -10686.852} C_VEL
LIN {X 0,Y 411.215,Z 304.258,A -85,B 0,C 180,E1 -10690.05,E2 -10690.05} C_VEL
LIN {X 0,Y 411.264,Z 304.256,A -85,B 0,C 180,E1 -10693.13,E2 -10693.13} C_VEL
LIN {X 0,Y 411.306,Z 304.252,A -85,B 0,C 180,E1 -10696.895,E2 -10696.895} C_VEL
LIN {X 0,Y 411.304,Z 304.25,A -85,B 0,C 180,E1 -10700.657,E2 -10700.657} C_VEL
LIN {X 0,Y 411.314,Z 304.299,A -85,B 0,C 180,E1 -10701.091,E2 -10701.091} C_VEL
LIN {X 0,Y 412.883,Z 313.047,A -85,B 0,C 180,E1 -10703.156,E2 -10703.156} C_VEL
LIN {X 0,Y 412.682,Z 321.455,A -85,B 0,C 180,E1 -10705.023,E2 -10705.023} C_VEL
LIN {X 0,Y 416.59,Z 342.836,A -85,B 0,C 180,E1 -10705.578,E2 -10705.578} C_VEL
LIN {X 0,Y 415.541,Z 429.113,A -85,B 0,C 180,E1 -10707.091,E2 -10707.091} C_VEL
LIN {X 0,Y 415.157,Z 441.701,A -85,B 0,C 180,E1 -10707.493,E2 -10707.493} C_VEL
LIN {X 0,Y 414.679,Z 454.758,A -85,B 0,C 180,E1 -10708.117,E2 -10708.117} C_VEL
LIN {X 0,Y 414.153,Z 464.405,A -85,B 0,C 180,E1 -10708.731,E2 -10708.731} C_VEL
LIN {X 0,Y 413.209,Z 469.632,A -85,B 0,C 180,E1 -10709.094,E2 -10709.094} C_VEL
LIN {X 0,Y 409.851,Z 477.864,A -85,B 0,C 180,E1 -10709.713,E2 -10709.713} C_VEL
LIN {X 0,Y 406.469,Z 485.633,A -85,B 0,C 180,E1 -10710.437,E2 -10710.437} C_VEL
LIN {X 0,Y 405.495,Z 490.129,A -85,B 0,C 180,E1 -10710.96,E2 -10710.96} C_VEL
LIN {X 0,Y 404.798,Z 499.375,A -85,B 0,C 180,E1 -10712.238,E2 -10712.238} C_VEL
LIN {X 0,Y 404.145,Z 508.164,A -85,B 0,C 180,E1 -10713.738,E2 -10713.738} C_VEL
LIN {X 0,Y 403.602,Z 515.2,A -85,B 0,C 180,E1 -10715.244,E2 -10715.244} C_VEL
LIN {X 0,Y 403.381,Z 520.756,A -85,B 0,C 180,E1 -10716.738,E2 -10716.738} C_VEL
LIN {X 0,Y 403.075,Z 525.861,A -85,B 0,C 180,E1 -10718.522,E2 -10718.522} C_VEL
LIN {X 0,Y 402.876,Z 529.038,A -85,B 0,C 180,E1 -10720.045,E2 -10720.045} C_VEL
LIN {X 0,Y 402.849,Z 530.616,A -85,B 0,C 180,E1 -10721.063,E2 -10721.063} C_VEL
LIN {X 0,Y 402.811,Z 531.915,A -85,B 0,C 180,E1 -10722.298,E2 -10722.298} C_VEL
LIN {X 0,Y 402.697,Z 532.761,A -85,B 0,C 180,E1 -10724.141,E2 -10724.141} C_VEL
LIN {X 0,Y 402.733,Z 532.663,A -85,B 0,C 180,E1 -10725.174,E2 -10725.174} C_VEL
LIN {X 0,Y 402.789,Z 532.008,A -85,B 0,C 180,E1 -10726.331,E2 -10726.331} C_VEL
LIN {X 0,Y 402.923,Z 529.738,A -85,B 0,C 180,E1 -10728.297,E2 -10728.297} C_VEL
LIN {X 0,Y 403.182,Z 527.037,A -85,B 0,C 180,E1 -10729.731,E2 -10729.731} C_VEL
LIN {X 0,Y 403.515,Z 522.611,A -85,B 0,C 180,E1 -10731.453,E2 -10731.453} C_VEL
LIN {X 0,Y 404.088,Z 516.097,A -85,B 0,C 180,E1 -10733.312,E2 -10733.312} C_VEL
LIN {X 0,Y 404.748,Z 509.039,A -85,B 0,C 180,E1 -10734.882,E2 -10734.882} C_VEL
LIN {X 0,Y 405.46,Z 501.522,A -85,B 0,C 180,E1 -10736.23,E2 -10736.23} C_VEL
LIN {X 0,Y 406.33,Z 491.337,A -85,B 0,C 180,E1 -10737.698,E2 -10737.698} C_VEL
LIN {X 0,Y 407.305,Z 480.99,A -85,B 0,C 180,E1 -10738.889,E2 -10738.889} C_VEL
LIN {X 0,Y 408.168,Z 471.015,A -85,B 0,C 180,E1 -10739.812,E2 -10739.812} C_VEL
LIN {X 0,Y 408.876,Z 460.221,A -85,B 0,C 180,E1 -10740.614,E2 -10740.614} C_VEL
LIN {X 0,Y 409.598,Z 447.274,A -85,B 0,C 180,E1 -10741.338,E2 -10741.338} C_VEL
LIN {X 0,Y 410.14,Z 434.667,A -85,B 0,C 180,E1 -10741.832,E2 -10741.832} C_VEL
LIN {X 0,Y 410.429,Z 420.88,A -85,B 0,C 180,E1 -10742.156,E2 -10742.156} C_VEL
LIN {X 0,Y 411.586,Z 343.492,A -85,B 0,C 180,E1 -10743.532,E2 -10743.532} C_VEL
LIN {X 0,Y 407.036,Z 323.189,A -85,B 0,C 180,E1 -10744.185,E2 -10744.185} C_VEL
LIN {X 0,Y 406.727,Z 321.513,A -85,B 0,C 180,E1 -10744.279,E2 -10744.279} C_VEL
LIN {X 0,Y 406.648,Z 316.97,A -85,B 0,C 180,E1 -10745.31,E2 -10745.31} C_VEL
LIN {X 0,Y 404.153,Z 305.145,A -85,B 0,C 180,E1 -10748.263,E2 -10748.263} C_VEL
LIN {X 0,Y 404.106,Z 305.145,A -85,B 0,C 180,E1 -10751.597,E2 -10751.597} C_VEL
LIN {X 0,Y 404.138,Z 305.145,A -85,B 0,C 180,E1 -10754.521,E2 -10754.521} C_VEL
LIN {X 0,Y 404.116,Z 305.141,A -85,B 0,C 180,E1 -10757.293,E2 -10757.293} C_VEL
LIN {X 0,Y 404.124,Z 305.143,A -85,B 0,C 180,E1 -10759.95,E2 -10759.95} C_VEL
LIN {X 0,Y 404.127,Z 305.146,A -85,B 0,C 180,E1 -10763.125,E2 -10763.125} C_VEL
LIN {X 0,Y 404.13,Z 305.128,A -85,B 0,C 180,E1 -10766.187,E2 -10766.187} C_VEL
LIN {X 0,Y 404.136,Z 305.143,A -85,B 0,C 180,E1 -10769.714,E2 -10769.714} C_VEL
LIN {X 0,Y 404.12,Z 305.145,A -85,B 0,C 180,E1 -10773.118,E2 -10773.118} C_VEL
LIN {X 0,Y 404.139,Z 305.141,A -85,B 0,C 180,E1 -10776.424,E2 -10776.424} C_VEL
LIN {X 0,Y 404.182,Z 305.141,A -85,B 0,C 180,E1 -10779.874,E2 -10779.874} C_VEL
LIN {X 0,Y 404.164,Z 305.134,A -85,B 0,C 180,E1 -10783.013,E2 -10783.013} C_VEL
LIN {X 0,Y 404.274,Z 305.117,A -85,B 0,C 180,E1 -10786.939,E2 -10786.939} C_VEL
LIN {X 0,Y 404.232,Z 305.132,A -85,B 0,C 180,E1 -10789.988,E2 -10789.988} C_VEL
LIN {X 0,Y 404.326,Z 305.115,A -85,B 0,C 180,E1 -10793.012,E2 -10793.012} C_VEL
LIN {X 0,Y 404.243,Z 305.125,A -85,B 0,C 180,E1 -10795.013,E2 -10795.013} C_VEL
LIN {X 0,Y 404.458,Z 305.097,A -85,B 0,C 180,E1 -10798.009,E2 -10798.009} C_VEL
LIN {X 0,Y 404.459,Z 305.096,A -85,B 0,C 180,E1 -10801.992,E2 -10801.992} C_VEL
LIN {X 0,Y 404.384,Z 305.11,A -85,B 0,C 180,E1 -10805.986,E2 -10805.986} C_VEL
LIN {X 0,Y 404.25,Z 305.127,A -85,B 0,C 180,E1 -10809.002,E2 -10809.002} C_VEL
LIN {X 0,Y 404.245,Z 305.123,A -85,B 0,C 180,E1 -10812.042,E2 -10812.042} C_VEL
LIN {X 0,Y 404.194,Z 305.136,A -85,B 0,C 180,E1 -10815.119,E2 -10815.119} C_VEL
LIN {X 0,Y 404.195,Z 305.124,A -85,B 0,C 180,E1 -10818.239,E2 -10818.239} C_VEL
LIN {X 0,Y 404.13,Z 305.141,A -85,B 0,C 180,E1 -10821.42,E2 -10821.42} C_VEL
LIN {X 0,Y 404.14,Z 305.139,A -85,B 0,C 180,E1 -10824.668,E2 -10824.668} C_VEL
LIN {X 0,Y 404.122,Z 305.14,A -85,B 0,C 180,E1 -10828.005,E2 -10828.005} C_VEL
LIN {X 0,Y 404.137,Z 305.14,A -85,B 0,C 180,E1 -10830.286,E2 -10830.286} C_VEL
LIN {X 0,Y 404.139,Z 305.143,A -85,B 0,C 180,E1 -10833.813,E2 -10833.813} C_VEL
LIN {X 0,Y 404.128,Z 305.142,A -85,B 0,C 180,E1 -10836.875,E2 -10836.875} C_VEL
LIN {X 0,Y 404.112,Z 305.148,A -85,B 0,C 180,E1 -10840.076,E2 -10840.076} C_VEL
LIN {X 0,Y 404.144,Z 305.13,A -85,B 0,C 180,E1 -10843.084,E2 -10843.084} C_VEL
LIN {X 0,Y 404.143,Z 305.149,A -85,B 0,C 180,E1 -10845.927,E2 -10845.927} C_VEL
LIN {X 0,Y 404.111,Z 305.149,A -85,B 0,C 180,E1 -10848.635,E2 -10848.635} C_VEL
LIN {X 0,Y 404.144,Z 305.145,A -85,B 0,C 180,E1 -10851.494,E2 -10851.494} C_VEL
LIN {X 0,Y 404.181,Z 305.134,A -85,B 0,C 180,E1 -10854.985,E2 -10854.985} C_VEL
LIN {X 0,Y 404.14,Z 305.144,A -85,B 0,C 180,E1 -10858.555,E2 -10858.555} C_VEL
LIN {X 0,Y 404.23,Z 305.303,A -85,B 0,C 180,E1 -10861.58,E2 -10861.58} C_VEL
LIN {X 0,Y 406.481,Z 315.559,A -85,B 0,C 180,E1 -10864.037,E2 -10864.037} C_VEL
LIN {X 0,Y 407.782,Z 323.572,A -85,B 0,C 180,E1 -10865.871,E2 -10865.871} C_VEL
LIN {X 0,Y 406.45,Z 340.38,A -85,B 0,C 180,E1 -10869.367,E2 -10869.367} C_VEL
LIN {X 0,Y 406.284,Z 342.447,A -85,B 0,C 180,E1 -10869.792,E2 -10869.792} C_VEL
LIN {X 0,Y 410.42,Z 364.445,A -85,B 0,C 180,E1 -10870.451,E2 -10870.451} C_VEL
LIN {X 0,Y 411.281,Z 371.202,A -85,B 0,C 180,E1 -10870.626,E2 -10870.626} C_VEL
LIN {X 0,Y 410.197,Z 450.839,A -85,B 0,C 180,E1 -10872.071,E2 -10872.071} C_VEL
LIN {X 0,Y 409.506,Z 464,A -85,B 0,C 180,E1 -10872.491,E2 -10872.491} C_VEL
LIN {X 0,Y 408.805,Z 477.19,A -85,B 0,C 180,E1 -10873.137,E2 -10873.137} C_VEL
LIN {X 0,Y 407.938,Z 488.318,A -85,B 0,C 180,E1 -10873.872,E2 -10873.872} C_VEL
LIN {X 0,Y 406.993,Z 499.882,A -85,B 0,C 180,E1 -10874.861,E2 -10874.861} C_VEL
LIN {X 0,Y 406.061,Z 510.306,A -85,B 0,C 180,E1 -10875.978,E2 -10875.978} C_VEL
LIN {X 0,Y 405.309,Z 519.716,A -85,B 0,C 180,E1 -10877.228,E2 -10877.228} C_VEL
LIN {X 0,Y 404.387,Z 528.802,A -85,B 0,C 180,E1 -10878.726,E2 -10878.726} C_VEL
LIN {X 0,Y 403.786,Z 536.141,A -85,B 0,C 180,E1 -10880.231,E2 -10880.231} C_VEL
LIN {X 0,Y 403.29,Z 542.901,A -85,B 0,C 180,E1 -10881.987,E2 -10881.987} C_VEL
LIN {X 0,Y 402.94,Z 548.19,A -85,B 0,C 180,E1 -10883.819,E2 -10883.819} C_VEL
LIN {X 0,Y 402.931,Z 550.785,A -85,B 0,C 180,E1 -10884.998,E2 -10884.998} C_VEL
LIN {X 0,Y 402.823,Z 553.783,A -85,B 0,C 180,E1 -10887.001,E2 -10887.001} C_VEL
LIN {X 0,Y 402.864,Z 554.693,A -85,B 0,C 180,E1 -10888.001,E2 -10888.001} C_VEL
LIN {X 0,Y 402.862,Z 555.182,A -85,B 0,C 180,E1 -10889.001,E2 -10889.001} C_VEL
LIN {X 0,Y 402.863,Z 554.946,A -85,B 0,C 180,E1 -10891,E2 -10891} C_VEL
LIN {X 0,Y 402.88,Z 554.25,A -85,B 0,C 180,E1 -10892,E2 -10892} C_VEL
LIN {X 0,Y 402.828,Z 553.132,A -85,B 0,C 180,E1 -10893.001,E2 -10893.001} C_VEL
LIN {X 0,Y 402.853,Z 551.573,A -85,B 0,C 180,E1 -10894.002,E2 -10894.002} C_VEL
LIN {X 0,Y 402.916,Z 548.432,A -85,B 0,C 180,E1 -10895.506,E2 -10895.506} C_VEL
LIN {X 0,Y 403.078,Z 544.219,A -85,B 0,C 180,E1 -10897.011,E2 -10897.011} C_VEL
LIN {X 0,Y 403.402,Z 537.795,A -85,B 0,C 180,E1 -10898.769,E2 -10898.769} C_VEL
LIN {X 0,Y 403.814,Z 530.776,A -85,B 0,C 180,E1 -10900.277,E2 -10900.277} C_VEL
LIN {X 0,Y 404.433,Z 521.964,A -85,B 0,C 180,E1 -10901.783,E2 -10901.783} C_VEL
LIN {X 0,Y 405.102,Z 512.931,A -85,B 0,C 180,E1 -10903.035,E2 -10903.035} C_VEL
LIN {X 0,Y 405.727,Z 503.931,A -85,B 0,C 180,E1 -10904.061,E2 -10904.061} C_VEL
LIN {X 0,Y 406.425,Z 493.502,A -85,B 0,C 180,E1 -10905.034,E2 -10905.034} C_VEL
LIN {X 0,Y 407.181,Z 481.589,A -85,B 0,C 180,E1 -10905.904,E2 -10905.904} C_VEL
LIN {X 0,Y 407.819,Z 469.176,A -85,B 0,C 180,E1 -10906.585,E2 -10906.585} C_VEL
LIN {X 0,Y 408.421,Z 456.45,A -85,B 0,C 180,E1 -10907.075,E2 -10907.075} C_VEL
LIN {X 0,Y 408.688,Z 443.067,A -85,B 0,C 180,E1 -10907.386,E2 -10907.386} C_VEL
LIN {X 0,Y 409.408,Z 368.632,A -85,B 0,C 180,E1 -10908.697,E2 -10908.697} C_VEL
LIN {X 0,Y 405.55,Z 342.841,A -85,B 0,C 180,E1 -10909.323,E2 -10909.323} C_VEL
LIN {X 0,Y 406.677,Z 325.344,A -85,B 0,C 180,E1 -10912.883,E2 -10912.883} C_VEL
LIN {X 0,Y 406.935,Z 319.689,A -85,B 0,C 180,E1 -10914.049,E2 -10914.049} C_VEL
LIN {X 0,Y 404.226,Z 305.135,A -85,B 0,C 180,E1 -10917.295,E2 -10917.295} C_VEL
LIN {X 0,Y 404.15,Z 305.14,A -85,B 0,C 180,E1 -10920.286,E2 -10920.286} C_VEL
LIN {X 0,Y 404.149,Z 305.144,A -85,B 0,C 180,E1 -10923.813,E2 -10923.813} C_VEL
LIN {X 0,Y 404.139,Z 305.139,A -85,B 0,C 180,E1 -10926.875,E2 -10926.875} C_VEL
LIN {X 0,Y 404.121,Z 305.148,A -85,B 0,C 180,E1 -10930.075,E2 -10930.075} C_VEL
LIN {X 0,Y 404.154,Z 305.137,A -85,B 0,C 180,E1 -10933.083,E2 -10933.083} C_VEL
LIN {X 0,Y 404.152,Z 305.139,A -85,B 0,C 180,E1 -10935.926,E2 -10935.926} C_VEL
LIN {X 0,Y 404.12,Z 305.148,A -85,B 0,C 180,E1 -10938.635,E2 -10938.635} C_VEL
LIN {X 0,Y 404.152,Z 305.137,A -85,B 0,C 180,E1 -10941.493,E2 -10941.493} C_VEL
LIN {X 0,Y 404.188,Z 305.138,A -85,B 0,C 180,E1 -10944.984,E2 -10944.984} C_VEL
LIN {X 0,Y 404.146,Z 305.141,A -85,B 0,C 180,E1 -10948.554,E2 -10948.554} C_VEL
LIN {X 0,Y 404.171,Z 305.135,A -85,B 0,C 180,E1 -10951.998,E2 -10951.998} C_VEL
LIN {X 0,Y 404.168,Z 305.141,A -85,B 0,C 180,E1 -10955.333,E2 -10955.333} C_VEL
LIN {X 0,Y 404.142,Z 305.139,A -85,B 0,C 180,E1 -10958.581,E2 -10958.581} C_VEL
LIN {X 0,Y 404.209,Z 305.134,A -85,B 0,C 180,E1 -10961.762,E2 -10961.762} C_VEL
LIN {X 0,Y 404.21,Z 305.131,A -85,B 0,C 180,E1 -10964.882,E2 -10964.882} C_VEL
LIN {X 0,Y 404.259,Z 305.128,A -85,B 0,C 180,E1 -10967.958,E2 -10967.958} C_VEL
LIN {X 0,Y 404.268,Z 305.123,A -85,B 0,C 180,E1 -10970.998,E2 -10970.998} C_VEL
LIN {X 0,Y 404.414,Z 305.111,A -85,B 0,C 180,E1 -10974.015,E2 -10974.015} C_VEL
LIN {X 0,Y 404.48,Z 305.104,A -85,B 0,C 180,E1 -10978.008,E2 -10978.008} C_VEL
LIN {X 0,Y 404.608,Z 305.087,A -85,B 0,C 180,E1 -10980,E2 -10980} C_VEL
LIN {X 0,Y 404.41,Z 305.106,A -85,B 0,C 180,E1 -10982.988,E2 -10982.988} C_VEL
LIN {X 0,Y 404.348,Z 305.113,A -85,B 0,C 180,E1 -10986.541,E2 -10986.541} C_VEL
LIN {X 0,Y 404.269,Z 305.124,A -85,B 0,C 180,E1 -10989.001,E2 -10989.001} C_VEL
LIN {X 0,Y 404.259,Z 305.126,A -85,B 0,C 180,E1 -10992.041,E2 -10992.041} C_VEL
LIN {X 0,Y 404.21,Z 305.133,A -85,B 0,C 180,E1 -10995.118,E2 -10995.118} C_VEL
LIN {X 0,Y 404.208,Z 305.132,A -85,B 0,C 180,E1 -10998.238,E2 -10998.238} C_VEL
LIN {X 0,Y 404.141,Z 305.141,A -85,B 0,C 180,E1 -11001.419,E2 -11001.419} C_VEL
LIN {X 0,Y 404.167,Z 305.138,A -85,B 0,C 180,E1 -11004.666,E2 -11004.666} C_VEL
LIN {X 0,Y 404.17,Z 305.135,A -85,B 0,C 180,E1 -11008.001,E2 -11008.001} C_VEL
LIN {X 0,Y 404.142,Z 305.143,A -85,B 0,C 180,E1 -11011.557,E2 -11011.557} C_VEL
LIN {X 0,Y 404.185,Z 305.136,A -85,B 0,C 180,E1 -11015.016,E2 -11015.016} C_VEL
LIN {X 0,Y 404.15,Z 305.138,A -85,B 0,C 180,E1 -11018.757,E2 -11018.757} C_VEL
LIN {X 0,Y 404.121,Z 305.148,A -85,B 0,C 180,E1 -11021.598,E2 -11021.598} C_VEL
LIN {X 0,Y 404.147,Z 305.139,A -85,B 0,C 180,E1 -11024.521,E2 -11024.521} C_VEL
LIN {X 0,Y 404.134,Z 305.141,A -85,B 0,C 180,E1 -11027.294,E2 -11027.294} C_VEL
LIN {X 0,Y 404.136,Z 305.146,A -85,B 0,C 180,E1 -11029.951,E2 -11029.951} C_VEL
LIN {X 0,Y 404.136,Z 305.139,A -85,B 0,C 180,E1 -11033.125,E2 -11033.125} C_VEL
LIN {X 0,Y 404.147,Z 305.145,A -85,B 0,C 180,E1 -11036.187,E2 -11036.187} C_VEL
LIN {X 0,Y 404.146,Z 305.139,A -85,B 0,C 180,E1 -11039.714,E2 -11039.714} C_VEL
LIN {X 0,Y 404.152,Z 305.139,A -85,B 0,C 180,E1 -11043.119,E2 -11043.119} C_VEL
LIN {X 0,Y 404.166,Z 305.14,A -85,B 0,C 180,E1 -11046.425,E2 -11046.425} C_VEL
LIN {X 0,Y 404.192,Z 305.132,A -85,B 0,C 180,E1 -11049.874,E2 -11049.874} C_VEL
LIN {X 0,Y 404.217,Z 305.136,A -85,B 0,C 180,E1 -11052.992,E2 -11052.992} C_VEL
LIN {X 0,Y 404.284,Z 305.127,A -85,B 0,C 180,E1 -11056.938,E2 -11056.938} C_VEL
LIN {X 0,Y 404.314,Z 305.191,A -85,B 0,C 180,E1 -11060.904,E2 -11060.904} C_VEL
LIN {X 0,Y 405.886,Z 314.101,A -85,B 0,C 180,E1 -11063.037,E2 -11063.037} C_VEL
LIN {X 0,Y 405.746,Z 321.686,A -85,B 0,C 180,E1 -11064.751,E2 -11064.751} C_VEL
LIN {X 0,Y 409.774,Z 344.275,A -85,B 0,C 180,E1 -11065.331,E2 -11065.331} C_VEL
LIN {X 0,Y 408.69,Z 429.026,A -85,B 0,C 180,E1 -11066.839,E2 -11066.839} C_VEL
LIN {X 0,Y 408.295,Z 441.38,A -85,B 0,C 180,E1 -11067.234,E2 -11067.234} C_VEL
LIN {X 0,Y 407.841,Z 453.771,A -85,B 0,C 180,E1 -11067.825,E2 -11067.825} C_VEL
LIN {X 0,Y 407.157,Z 466.335,A -85,B 0,C 180,E1 -11068.639,E2 -11068.639} C_VEL
LIN {X 0,Y 406.397,Z 477.919,A -85,B 0,C 180,E1 -11069.628,E2 -11069.628} C_VEL
LIN {X 0,Y 405.635,Z 488.349,A -85,B 0,C 180,E1 -11070.744,E2 -11070.744} C_VEL
LIN {X 0,Y 405.495,Z 490.129,A -85,B 0,C 180,E1 -11070.96,E2 -11070.96} C_VEL
LIN {X 0,Y 404.541,Z 494.515,A -85,B 0,C 180,E1 -11071.515,E2 -11071.515} C_VEL
LIN {X 0,Y 401.208,Z 501.267,A -85,B 0,C 180,E1 -11072.437,E2 -11072.437} C_VEL
LIN {X 0,Y 397.877,Z 507.419,A -85,B 0,C 180,E1 -11073.441,E2 -11073.441} C_VEL
LIN {X 0,Y 396.935,Z 510.86,A -85,B 0,C 180,E1 -11074.114,E2 -11074.114} C_VEL
LIN {X 0,Y 396.501,Z 517.201,A -85,B 0,C 180,E1 -11075.594,E2 -11075.594} C_VEL
LIN {X 0,Y 396.232,Z 522.458,A -85,B 0,C 180,E1 -11077.131,E2 -11077.131} C_VEL
LIN {X 0,Y 395.98,Z 526.557,A -85,B 0,C 180,E1 -11078.676,E2 -11078.676} C_VEL
LIN {X 0,Y 395.774,Z 529.598,A -85,B 0,C 180,E1 -11080.228,E2 -11080.228} C_VEL
LIN {X 0,Y 395.736,Z 531.069,A -85,B 0,C 180,E1 -11081.264,E2 -11081.264} C_VEL
LIN {X 0,Y 395.706,Z 532.147,A -85,B 0,C 180,E1 -11082.357,E2 -11082.357} C_VEL
LIN {X 0,Y 395.599,Z 532.989,A -85,B 0,C 180,E1 -11084.4,E2 -11084.4} C_VEL
LIN {X 0,Y 395.658,Z 532.77,A -85,B 0,C 180,E1 -11085.452,E2 -11085.452} C_VEL
LIN {X 0,Y 395.709,Z 532.14,A -85,B 0,C 180,E1 -11086.508,E2 -11086.508} C_VEL
LIN {X 0,Y 395.774,Z 531.1,A -85,B 0,C 180,E1 -11087.569,E2 -11087.569} C_VEL
LIN {X 0,Y 395.891,Z 529.593,A -85,B 0,C 180,E1 -11088.634,E2 -11088.634} C_VEL
LIN {X 0,Y 396.201,Z 526.36,A -85,B 0,C 180,E1 -11090.274,E2 -11090.274} C_VEL
LIN {X 0,Y 396.544,Z 522.143,A -85,B 0,C 180,E1 -11091.849,E2 -11091.849} C_VEL
LIN {X 0,Y 397.087,Z 516.534,A -85,B 0,C 180,E1 -11093.465,E2 -11093.465} C_VEL
LIN {X 0,Y 397.789,Z 509.416,A -85,B 0,C 180,E1 -11095.088,E2 -11095.088} C_VEL
LIN {X 0,Y 398.543,Z 502.063,A -85,B 0,C 180,E1 -11096.439,E2 -11096.439} C_VEL
LIN {X 0,Y 399.388,Z 493.021,A -85,B 0,C 180,E1 -11097.794,E2 -11097.794} C_VEL
LIN {X 0,Y 400.337,Z 483.094,A -85,B 0,C 180,E1 -11098.996,E2 -11098.996} C_VEL
LIN {X 0,Y 401.377,Z 471.904,A -85,B 0,C 180,E1 -11100.079,E2 -11100.079} C_VEL
LIN {X 0,Y 402.16,Z 460.846,A -85,B 0,C 180,E1 -11100.925,E2 -11100.925} C_VEL
LIN {X 0,Y 402.925,Z 448.741,A -85,B 0,C 180,E1 -11101.624,E2 -11101.624} C_VEL
LIN {X 0,Y 403.487,Z 435.65,A -85,B 0,C 180,E1 -11102.163,E2 -11102.163} C_VEL
LIN {X 0,Y 403.828,Z 421.971,A -85,B 0,C 180,E1 -11102.501,E2 -11102.501} C_VEL
LIN {X 0,Y 405.028,Z 344.605,A -85,B 0,C 180,E1 -11103.9,E2 -11103.9} C_VEL
LIN {X 0,Y 400.42,Z 323.988,A -85,B 0,C 180,E1 -11104.582,E2 -11104.582} C_VEL
LIN {X 0,Y 399.907,Z 321.74,A -85,B 0,C 180,E1 -11104.696,E2 -11104.696} C_VEL
LIN {X 0,Y 399.753,Z 318.474,A -85,B 0,C 180,E1 -11105.461,E2 -11105.461} C_VEL
LIN {X 0,Y 397.105,Z 306.024,A -85,B 0,C 180,E1 -11108.609,E2 -11108.609} C_VEL
LIN {X 0,Y 397.054,Z 306.025,A -85,B 0,C 180,E1 -11112.267,E2 -11112.267} C_VEL
LIN {X 0,Y 397.079,Z 306.025,A -85,B 0,C 180,E1 -11115.068,E2 -11115.068} C_VEL
LIN {X 0,Y 397.046,Z 306.024,A -85,B 0,C 180,E1 -11118.023,E2 -11118.023} C_VEL
LIN {X 0,Y 397.086,Z 306.021,A -85,B 0,C 180,E1 -11121.723,E2 -11121.723} C_VEL
LIN {X 0,Y 397.111,Z 306.005,A -85,B 0,C 180,E1 -11125.506,E2 -11125.506} C_VEL
LIN {X 0,Y 397.069,Z 306.025,A -85,B 0,C 180,E1 -11129.117,E2 -11129.117} C_VEL
LIN {X 0,Y 397.09,Z 306.019,A -85,B 0,C 180,E1 -11132.602,E2 -11132.602} C_VEL
LIN {X 0,Y 397.102,Z 306.021,A -85,B 0,C 180,E1 -11135.98,E2 -11135.98} C_VEL
LIN {X 0,Y 397.13,Z 306.018,A -85,B 0,C 180,E1 -11139.704,E2 -11139.704} C_VEL
LIN {X 0,Y 397.144,Z 306.008,A -85,B 0,C 180,E1 -11142.858,E2 -11142.858} C_VEL
LIN {X 0,Y 397.22,Z 305.996,A -85,B 0,C 180,E1 -11146.703,E2 -11146.703} C_VEL
LIN {X 0,Y 397.194,Z 306.008,A -85,B 0,C 180,E1 -11149.809,E2 -11149.809} C_VEL
LIN {X 0,Y 397.28,Z 305.994,A -85,B 0,C 180,E1 -11152.887,E2 -11152.887} C_VEL
LIN {X 0,Y 397.214,Z 306.001,A -85,B 0,C 180,E1 -11154.925,E2 -11154.925} C_VEL
LIN {X 0,Y 397.426,Z 305.973,A -85,B 0,C 180,E1 -11157.973,E2 -11157.973} C_VEL
LIN {X 0,Y 397.427,Z 305.972,A -85,B 0,C 180,E1 -11162.027,E2 -11162.027} C_VEL
LIN {X 0,Y 397.337,Z 305.989,A -85,B 0,C 180,E1 -11166.092,E2 -11166.092} C_VEL
LIN {X 0,Y 397.221,Z 306.002,A -85,B 0,C 180,E1 -11169.163,E2 -11169.163} C_VEL
LIN {X 0,Y 397.209,Z 306.001,A -85,B 0,C 180,E1 -11172.259,E2 -11172.259} C_VEL
LIN {X 0,Y 397.168,Z 306.009,A -85,B 0,C 180,E1 -11175.393,E2 -11175.393} C_VEL
LIN {X 0,Y 397.149,Z 306.003,A -85,B 0,C 180,E1 -11178.574,E2 -11178.574} C_VEL
LIN {X 0,Y 397.087,Z 306.015,A -85,B 0,C 180,E1 -11181.819,E2 -11181.819} C_VEL
LIN {X 0,Y 397.09,Z 306.022,A -85,B 0,C 180,E1 -11185.136,E2 -11185.136} C_VEL
LIN {X 0,Y 397.07,Z 306.018,A -85,B 0,C 180,E1 -11188.548,E2 -11188.548} C_VEL
LIN {X 0,Y 397.075,Z 306.019,A -85,B 0,C 180,E1 -11191.837,E2 -11191.837} C_VEL
LIN {X 0,Y 397.119,Z 306.014,A -85,B 0,C 180,E1 -11194.494,E2 -11194.494} C_VEL
LIN {X 0,Y 397.086,Z 306.017,A -85,B 0,C 180,E1 -11198.277,E2 -11198.277} C_VEL
LIN {X 0,Y 397.053,Z 306.019,A -85,B 0,C 180,E1 -11201.979,E2 -11201.979} C_VEL
LIN {X 0,Y 397.082,Z 306.019,A -85,B 0,C 180,E1 -11205.07,E2 -11205.07} C_VEL
LIN {X 0,Y 397.058,Z 306.03,A -85,B 0,C 180,E1 -11208.023,E2 -11208.023} C_VEL
LIN {X 0,Y 397.12,Z 306.019,A -85,B 0,C 180,E1 -11211.141,E2 -11211.141} C_VEL
LIN {X 0,Y 397.116,Z 306.017,A -85,B 0,C 180,E1 -11214.498,E2 -11214.498} C_VEL
LIN {X 0,Y 397.076,Z 306.021,A -85,B 0,C 180,E1 -11217.93,E2 -11217.93} C_VEL
LIN {X 0,Y 397.158,Z 306.064,A -85,B 0,C 180,E1 -11221.172,E2 -11221.172} C_VEL
LIN {X 0,Y 399.644,Z 317.272,A -85,B 0,C 180,E1 -11223.92,E2 -11223.92} C_VEL
LIN {X 0,Y 400.901,Z 325.021,A -85,B 0,C 180,E1 -11225.726,E2 -11225.726} C_VEL
LIN {X 0,Y 399.555,Z 341.2,A -85,B 0,C 180,E1 -11229.154,E2 -11229.154} C_VEL
LIN {X 0,Y 399.48,Z 342.223,A -85,B 0,C 180,E1 -11229.369,E2 -11229.369} C_VEL
LIN {X 0,Y 403.797,Z 365.004,A -85,B 0,C 180,E1 -11230.074,E2 -11230.074} C_VEL
LIN {X 0,Y 404.702,Z 372.64,A -85,B 0,C 180,E1 -11230.273,E2 -11230.273} C_VEL
LIN {X 0,Y 403.58,Z 450.4,A -85,B 0,C 180,E1 -11231.704,E2 -11231.704} C_VEL
LIN {X 0,Y 402.888,Z 463.562,A -85,B 0,C 180,E1 -11232.128,E2 -11232.128} C_VEL
LIN {X 0,Y 402.122,Z 476.819,A -85,B 0,C 180,E1 -11232.782,E2 -11232.782} C_VEL
LIN {X 0,Y 401.16,Z 488.772,A -85,B 0,C 180,E1 -11233.592,E2 -11233.592} C_VEL
LIN {X 0,Y 400.144,Z 500.206,A -85,B 0,C 180,E1 -11234.595,E2 -11234.595} C_VEL
LIN {X 0,Y 399.163,Z 510.529,A -85,B 0,C 180,E1 -11235.731,E2 -11235.731} C_VEL
LIN {X 0,Y 398.369,Z 519.833,A -85,B 0,C 180,E1 -11237.002,E2 -11237.002} C_VEL
LIN {X 0,Y 397.417,Z 528.854,A -85,B 0,C 180,E1 -11238.526,E2 -11238.526} C_VEL
LIN {X 0,Y 396.757,Z 536.148,A -85,B 0,C 180,E1 -11240.056,E2 -11240.056} C_VEL
LIN {X 0,Y 396.235,Z 542.85,A -85,B 0,C 180,E1 -11241.843,E2 -11241.843} C_VEL
LIN {X 0,Y 395.937,Z 547.293,A -85,B 0,C 180,E1 -11243.376,E2 -11243.376} C_VEL
LIN {X 0,Y 395.844,Z 550.668,A -85,B 0,C 180,E1 -11244.908,E2 -11244.908} C_VEL
LIN {X 0,Y 395.775,Z 552.352,A -85,B 0,C 180,E1 -11245.928,E2 -11245.928} C_VEL
LIN {X 0,Y 395.762,Z 554.529,A -85,B 0,C 180,E1 -11247.966,E2 -11247.966} C_VEL
LIN {X 0,Y 395.791,Z 554.99,A -85,B 0,C 180,E1 -11248.983,E2 -11248.983} C_VEL
LIN {X 0,Y 395.792,Z 554.726,A -85,B 0,C 180,E1 -11251.018,E2 -11251.018} C_VEL
LIN {X 0,Y 395.778,Z 554.013,A -85,B 0,C 180,E1 -11252.036,E2 -11252.036} C_VEL
LIN {X 0,Y 395.731,Z 552.864,A -85,B 0,C 180,E1 -11253.055,E2 -11253.055} C_VEL
LIN {X 0,Y 395.776,Z 551.289,A -85,B 0,C 180,E1 -11254.074,E2 -11254.074} C_VEL
LIN {X 0,Y 395.827,Z 547.623,A -85,B 0,C 180,E1 -11255.805,E2 -11255.805} C_VEL
LIN {X 0,Y 396.065,Z 542.215,A -85,B 0,C 180,E1 -11257.649,E2 -11257.649} C_VEL
LIN {X 0,Y 396.468,Z 535.194,A -85,B 0,C 180,E1 -11259.438,E2 -11259.438} C_VEL
LIN {X 0,Y 396.961,Z 527.586,A -85,B 0,C 180,E1 -11260.973,E2 -11260.973} C_VEL
LIN {X 0,Y 397.6,Z 519.81,A -85,B 0,C 180,E1 -11262.247,E2 -11262.247} C_VEL
LIN {X 0,Y 398.334,Z 510.741,A -85,B 0,C 180,E1 -11263.468,E2 -11263.468} C_VEL
LIN {X 0,Y 399.001,Z 499.723,A -85,B 0,C 180,E1 -11264.668,E2 -11264.668} C_VEL
LIN {X 0,Y 399.858,Z 487.958,A -85,B 0,C 180,E1 -11265.679,E2 -11265.679} C_VEL
LIN {X 0,Y 400.669,Z 475.367,A -85,B 0,C 180,E1 -11266.496,E2 -11266.496} C_VEL
LIN {X 0,Y 401.262,Z 462.822,A -85,B 0,C 180,E1 -11267.094,E2 -11267.094} C_VEL
LIN {X 0,Y 401.728,Z 449.935,A -85,B 0,C 180,E1 -11267.5,E2 -11267.5} C_VEL
LIN {X 0,Y 402.603,Z 369.522,A -85,B 0,C 180,E1 -11268.953,E2 -11268.953} C_VEL
LIN {X 0,Y 398.592,Z 342.538,A -85,B 0,C 180,E1 -11269.641,E2 -11269.641} C_VEL
LIN {X 0,Y 399.698,Z 326.159,A -85,B 0,C 180,E1 -11273.032,E2 -11273.032} C_VEL
LIN {X 0,Y 399.972,Z 321.637,A -85,B 0,C 180,E1 -11273.977,E2 -11273.977} C_VEL
LIN {X 0,Y 397.789,Z 309.124,A -85,B 0,C 180,E1 -11276.778,E2 -11276.778} C_VEL
LIN {X 0,Y 397.201,Z 306.01,A -85,B 0,C 180,E1 -11277.534,E2 -11277.534} C_VEL
LIN {X 0,Y 397.083,Z 306.018,A -85,B 0,C 180,E1 -11280.883,E2 -11280.883} C_VEL
LIN {X 0,Y 397.13,Z 306.014,A -85,B 0,C 180,E1 -11284.494,E2 -11284.494} C_VEL
LIN {X 0,Y 397.096,Z 306.022,A -85,B 0,C 180,E1 -11288.277,E2 -11288.277} C_VEL
LIN {X 0,Y 397.062,Z 306.025,A -85,B 0,C 180,E1 -11291.978,E2 -11291.978} C_VEL
LIN {X 0,Y 397.091,Z 306.018,A -85,B 0,C 180,E1 -11295.069,E2 -11295.069} C_VEL
LIN {X 0,Y 397.066,Z 306.022,A -85,B 0,C 180,E1 -11298.022,E2 -11298.022} C_VEL
LIN {X 0,Y 397.128,Z 306.014,A -85,B 0,C 180,E1 -11301.14,E2 -11301.14} C_VEL
LIN {X 0,Y 397.123,Z 306.017,A -85,B 0,C 180,E1 -11304.497,E2 -11304.497} C_VEL
LIN {X 0,Y 397.082,Z 306.018,A -85,B 0,C 180,E1 -11307.928,E2 -11307.928} C_VEL
LIN {X 0,Y 397.103,Z 306.018,A -85,B 0,C 180,E1 -11311.455,E2 -11311.455} C_VEL
LIN {X 0,Y 397.127,Z 306.017,A -85,B 0,C 180,E1 -11314.866,E2 -11314.866} C_VEL
LIN {X 0,Y 397.1,Z 306.016,A -85,B 0,C 180,E1 -11318.181,E2 -11318.181} C_VEL
LIN {X 0,Y 397.162,Z 306.016,A -85,B 0,C 180,E1 -11321.426,E2 -11321.426} C_VEL
LIN {X 0,Y 397.183,Z 306.005,A -85,B 0,C 180,E1 -11324.608,E2 -11324.608} C_VEL
LIN {X 0,Y 397.223,Z 306.007,A -85,B 0,C 180,E1 -11327.742,E2 -11327.742} C_VEL
LIN {X 0,Y 397.238,Z 305.999,A -85,B 0,C 180,E1 -11330.838,E2 -11330.838} C_VEL
LIN {X 0,Y 397.364,Z 305.99,A -85,B 0,C 180,E1 -11333.908,E2 -11333.908} C_VEL
LIN {X 0,Y 397.448,Z 305.98,A -85,B 0,C 180,E1 -11337.973,E2 -11337.973} C_VEL
LIN {X 0,Y 397.578,Z 305.963,A -85,B 0,C 180,E1 -11340,E2 -11340} C_VEL
LIN {X 0,Y 397.344,Z 305.986,A -85,B 0,C 180,E1 -11343.041,E2 -11343.041} C_VEL
LIN {X 0,Y 397.304,Z 305.991,A -85,B 0,C 180,E1 -11346.534,E2 -11346.534} C_VEL
LIN {X 0,Y 397.239,Z 305.999,A -85,B 0,C 180,E1 -11349.162,E2 -11349.162} C_VEL
LIN {X 0,Y 397.222,Z 306.004,A -85,B 0,C 180,E1 -11352.258,E2 -11352.258} C_VEL
LIN {X 0,Y 397.183,Z 306.006,A -85,B 0,C 180,E1 -11355.392,E2 -11355.392} C_VEL
LIN {X 0,Y 397.161,Z 306.013,A -85,B 0,C 180,E1 -11358.573,E2 -11358.573} C_VEL
LIN {X 0,Y 397.099,Z 306.016,A -85,B 0,C 180,E1 -11361.818,E2 -11361.818} C_VEL
LIN {X 0,Y 397.126,Z 306.02,A -85,B 0,C 180,E1 -11365.133,E2 -11365.133} C_VEL
LIN {X 0,Y 397.101,Z 306.017,A -85,B 0,C 180,E1 -11368.545,E2 -11368.545} C_VEL
LIN {X 0,Y 397.08,Z 306.019,A -85,B 0,C 180,E1 -11372.071,E2 -11372.071} C_VEL
LIN {X 0,Y 397.121,Z 306.021,A -85,B 0,C 180,E1 -11375.503,E2 -11375.503} C_VEL
LIN {X 0,Y 397.126,Z 306.013,A -85,B 0,C 180,E1 -11378.86,E2 -11378.86} C_VEL
LIN {X 0,Y 397.067,Z 306.022,A -85,B 0,C 180,E1 -11382.267,E2 -11382.267} C_VEL
LIN {X 0,Y 397.088,Z 306.018,A -85,B 0,C 180,E1 -11385.068,E2 -11385.068} C_VEL
LIN {X 0,Y 397.063,Z 306.027,A -85,B 0,C 180,E1 -11388.021,E2 -11388.021} C_VEL
LIN {X 0,Y 397.104,Z 306.015,A -85,B 0,C 180,E1 -11391.143,E2 -11391.143} C_VEL
LIN {X 0,Y 397.121,Z 306.017,A -85,B 0,C 180,E1 -11394.496,E2 -11394.496} C_VEL
LIN {X 0,Y 397.08,Z 306.021,A -85,B 0,C 180,E1 -11397.928,E2 -11397.928} C_VEL
LIN {X 0,Y 397.1,Z 306.016,A -85,B 0,C 180,E1 -11401.454,E2 -11401.454} C_VEL
LIN {X 0,Y 397.125,Z 306.017,A -85,B 0,C 180,E1 -11404.865,E2 -11404.865} C_VEL
LIN {X 0,Y 397.098,Z 306.018,A -85,B 0,C 180,E1 -11408.181,E2 -11408.181} C_VEL
LIN {X 0,Y 397.159,Z 306.01,A -85,B 0,C 180,E1 -11411.426,E2 -11411.426} C_VEL
LIN {X 0,Y 397.179,Z 306.009,A -85,B 0,C 180,E1 -11414.607,E2 -11414.607} C_VEL
LIN {X 0,Y 397.219,Z 306.002,A -85,B 0,C 180,E1 -11417.741,E2 -11417.741} C_VEL
LIN {X 0,Y 397.258,Z 306.104,A -85,B 0,C 180,E1 -11420.709,E2 -11420.709} C_VEL
LIN {X 0,Y 398.888,Z 315.151,A -85,B 0,C 180,E1 -11422.915,E2 -11422.915} C_VEL
LIN {X 0,Y 398.828,Z 321.778,A -85,B 0,C 180,E1 -11424.438,E2 -11424.438} C_VEL
LIN {X 0,Y 402.968,Z 344.655,A -85,B 0,C 180,E1 -11425.059,E2 -11425.059} C_VEL
LIN {X 0,Y 401.821,Z 429.524,A -85,B 0,C 180,E1 -11426.595,E2 -11426.595} C_VEL
LIN {X 0,Y 401.411,Z 442.24,A -85,B 0,C 180,E1 -11427.017,E2 -11427.017} C_VEL
LIN {X 0,Y 400.91,Z 454.978,A -85,B 0,C 180,E1 -11427.645,E2 -11427.645} C_VEL
LIN {X 0,Y 400.18,Z 467.456,A -85,B 0,C 180,E1 -11428.49,E2 -11428.49} C_VEL
LIN {X 0,Y 399.404,Z 478.87,A -85,B 0,C 180,E1 -11429.495,E2 -11429.495} C_VEL
LIN {X 0,Y 398.616,Z 489.172,A -85,B 0,C 180,E1 -11430.63,E2 -11430.63} C_VEL
LIN {X 0,Y 397.996,Z 497.586,A -85,B 0,C 180,E1 -11431.77,E2 -11431.77} C_VEL
LIN {X 0,Y 397.239,Z 506.725,A -85,B 0,C 180,E1 -11433.295,E2 -11433.295} C_VEL
LIN {X 0,Y 396.935,Z 510.86,A -85,B 0,C 180,E1 -11434.114,E2 -11434.114} C_VEL
LIN {X 0,Y 396.036,Z 514.129,A -85,B 0,C 180,E1 -11434.814,E2 -11434.814} C_VEL
LIN {X 0,Y 392.896,Z 518.976,A -85,B 0,C 180,E1 -11435.986,E2 -11435.986} C_VEL
LIN {X 0,Y 389.799,Z 523.125,A -85,B 0,C 180,E1 -11437.229,E2 -11437.229} C_VEL
LIN {X 0,Y 388.984,Z 525.301,A -85,B 0,C 180,E1 -11438.031,E2 -11438.031} C_VEL
LIN {X 0,Y 388.787,Z 528.29,A -85,B 0,C 180,E1 -11439.362,E2 -11439.362} C_VEL
LIN {X 0,Y 388.681,Z 530.122,A -85,B 0,C 180,E1 -11440.416,E2 -11440.416} C_VEL
LIN {X 0,Y 388.616,Z 532.385,A -85,B 0,C 180,E1 -11442.427,E2 -11442.427} C_VEL
LIN {X 0,Y 388.535,Z 533.044,A -85,B 0,C 180,E1 -11443.599,E2 -11443.599} C_VEL
LIN {X 0,Y 388.506,Z 533.165,A -85,B 0,C 180,E1 -11444.669,E2 -11444.669} C_VEL
LIN {X 0,Y 388.615,Z 532.368,A -85,B 0,C 180,E1 -11446.567,E2 -11446.567} C_VEL
LIN {X 0,Y 388.732,Z 531.042,A -85,B 0,C 180,E1 -11447.898,E2 -11447.898} C_VEL
LIN {X 0,Y 388.979,Z 528.479,A -85,B 0,C 180,E1 -11449.526,E2 -11449.526} C_VEL
LIN {X 0,Y 389.317,Z 524.814,A -85,B 0,C 180,E1 -11451.163,E2 -11451.163} C_VEL
LIN {X 0,Y 389.767,Z 520.234,A -85,B 0,C 180,E1 -11452.716,E2 -11452.716} C_VEL
LIN {X 0,Y 390.465,Z 513.642,A -85,B 0,C 180,E1 -11454.454,E2 -11454.454} C_VEL
LIN {X 0,Y 391.243,Z 505.849,A -85,B 0,C 180,E1 -11456.083,E2 -11456.083} C_VEL
LIN {X 0,Y 392.161,Z 497.477,A -85,B 0,C 180,E1 -11457.481,E2 -11457.481} C_VEL
LIN {X 0,Y 393.097,Z 488.368,A -85,B 0,C 180,E1 -11458.722,E2 -11458.722} C_VEL
LIN {X 0,Y 394.162,Z 477.193,A -85,B 0,C 180,E1 -11459.949,E2 -11459.949} C_VEL
LIN {X 0,Y 395.132,Z 466.188,A -85,B 0,C 180,E1 -11460.902,E2 -11460.902} C_VEL
LIN {X 0,Y 395.979,Z 453.869,A -85,B 0,C 180,E1 -11461.721,E2 -11461.721} C_VEL
LIN {X 0,Y 396.63,Z 441.244,A -85,B 0,C 180,E1 -11462.336,E2 -11462.336} C_VEL
LIN {X 0,Y 397.118,Z 428.525,A -85,B 0,C 180,E1 -11462.742,E2 -11462.742} C_VEL
LIN {X 0,Y 398.495,Z 345.614,A -85,B 0,C 180,E1 -11464.283,E2 -11464.283} C_VEL
LIN {X 0,Y 394.166,Z 326.193,A -85,B 0,C 180,E1 -11464.944,E2 -11464.944} C_VEL
LIN {X 0,Y 393.089,Z 321.973,A -85,B 0,C 180,E1 -11465.132,E2 -11465.132} C_VEL
LIN {X 0,Y 391.46,Z 313.368,A -85,B 0,C 180,E1 -11467.294,E2 -11467.294} C_VEL
LIN {X 0,Y 390.035,Z 306.901,A -85,B 0,C 180,E1 -11469.002,E2 -11469.002} C_VEL
LIN {X 0,Y 390.029,Z 306.9,A -85,B 0,C 180,E1 -11472.372,E2 -11472.372} C_VEL
LIN {X 0,Y 390.036,Z 306.903,A -85,B 0,C 180,E1 -11475.353,E2 -11475.353} C_VEL
LIN {X 0,Y 390.009,Z 306.901,A -85,B 0,C 180,E1 -11478.184,E2 -11478.184} C_VEL
LIN {X 0,Y 390.052,Z 306.899,A -85,B 0,C 180,E1 -11480.903,E2 -11480.903} C_VEL
LIN {X 0,Y 390.073,Z 306.893,A -85,B 0,C 180,E1 -11484.792,E2 -11484.792} C_VEL
LIN {X 0,Y 390.014,Z 306.901,A -85,B 0,C 180,E1 -11488.495,E2 -11488.495} C_VEL
LIN {X 0,Y 390.028,Z 306.901,A -85,B 0,C 180,E1 -11492.063,E2 -11492.063} C_VEL
LIN {X 0,Y 390.034,Z 306.9,A -85,B 0,C 180,E1 -11495.516,E2 -11495.516} C_VEL
LIN {X 0,Y 390.046,Z 306.894,A -85,B 0,C 180,E1 -11498.877,E2 -11498.877} C_VEL
LIN {X 0,Y 390.059,Z 306.892,A -85,B 0,C 180,E1 -11502.164,E2 -11502.164} C_VEL
LIN {X 0,Y 390.081,Z 306.892,A -85,B 0,C 180,E1 -11505.39,E2 -11505.39} C_VEL
LIN {X 0,Y 390.157,Z 306.876,A -85,B 0,C 180,E1 -11507.517,E2 -11507.517} C_VEL
LIN {X 0,Y 390.175,Z 306.874,A -85,B 0,C 180,E1 -11510.671,E2 -11510.671} C_VEL
LIN {X 0,Y 390.261,Z 306.87,A -85,B 0,C 180,E1 -11513.797,E2 -11513.797} C_VEL
LIN {X 0,Y 390.392,Z 306.848,A -85,B 0,C 180,E1 -11517.937,E2 -11517.937} C_VEL
LIN {X 0,Y 390.393,Z 306.847,A -85,B 0,C 180,E1 -11522.064,E2 -11522.064} C_VEL
LIN {X 0,Y 390.293,Z 306.867,A -85,B 0,C 180,E1 -11526.203,E2 -11526.203} C_VEL
LIN {X 0,Y 390.179,Z 306.878,A -85,B 0,C 180,E1 -11529.33,E2 -11529.33} C_VEL
LIN {X 0,Y 390.161,Z 306.878,A -85,B 0,C 180,E1 -11532.484,E2 -11532.484} C_VEL
LIN {X 0,Y 390.129,Z 306.884,A -85,B 0,C 180,E1 -11535.678,E2 -11535.678} C_VEL
LIN {X 0,Y 390.094,Z 306.884,A -85,B 0,C 180,E1 -11538.923,E2 -11538.923} C_VEL
LIN {X 0,Y 390.027,Z 306.894,A -85,B 0,C 180,E1 -11542.235,E2 -11542.235} C_VEL
LIN {X 0,Y 390.042,Z 306.897,A -85,B 0,C 180,E1 -11545.723,E2 -11545.723} C_VEL
LIN {X 0,Y 390.026,Z 306.9,A -85,B 0,C 180,E1 -11549.113,E2 -11549.113} C_VEL
LIN {X 0,Y 390.037,Z 306.895,A -85,B 0,C 180,E1 -11552.722,E2 -11552.722} C_VEL
LIN {X 0,Y 390.049,Z 306.896,A -85,B 0,C 180,E1 -11555.826,E2 -11555.826} C_VEL
LIN {X 0,Y 390.032,Z 306.897,A -85,B 0,C 180,E1 -11559.213,E2 -11559.213} C_VEL
LIN {X 0,Y 390.031,Z 306.89,A -85,B 0,C 180,E1 -11562.374,E2 -11562.374} C_VEL
LIN {X 0,Y 390.039,Z 306.898,A -85,B 0,C 180,E1 -11565.355,E2 -11565.355} C_VEL
LIN {X 0,Y 390.024,Z 306.907,A -85,B 0,C 180,E1 -11568.187,E2 -11568.187} C_VEL
LIN {X 0,Y 390.079,Z 306.896,A -85,B 0,C 180,E1 -11570.908,E2 -11570.908} C_VEL
LIN {X 0,Y 390.082,Z 306.891,A -85,B 0,C 180,E1 -11574.794,E2 -11574.794} C_VEL
LIN {X 0,Y 390.022,Z 306.902,A -85,B 0,C 180,E1 -11578.497,E2 -11578.497} C_VEL
LIN {X 0,Y 390.12,Z 306.982,A -85,B 0,C 180,E1 -11580.786,E2 -11580.786} C_VEL
LIN {X 0,Y 392.576,Z 317.871,A -85,B 0,C 180,E1 -11583.524,E2 -11583.524} C_VEL
LIN {X 0,Y 393.994,Z 325.998,A -85,B 0,C 180,E1 -11585.469,E2 -11585.469} C_VEL
LIN {X 0,Y 393.062,Z 337.432,A -85,B 0,C 180,E1 -11587.947,E2 -11587.947} C_VEL
LIN {X 0,Y 392.68,Z 342.019,A -85,B 0,C 180,E1 -11588.931,E2 -11588.931} C_VEL
LIN {X 0,Y 397.201,Z 365.473,A -85,B 0,C 180,E1 -11589.682,E2 -11589.682} C_VEL
LIN {X 0,Y 398.156,Z 373.048,A -85,B 0,C 180,E1 -11589.888,E2 -11589.888} C_VEL
LIN {X 0,Y 396.94,Z 451.033,A -85,B 0,C 180,E1 -11591.355,E2 -11591.355} C_VEL
LIN {X 0,Y 396.169,Z 464.64,A -85,B 0,C 180,E1 -11591.815,E2 -11591.815} C_VEL
LIN {X 0,Y 395.389,Z 477.507,A -85,B 0,C 180,E1 -11592.48,E2 -11592.48} C_VEL
LIN {X 0,Y 394.386,Z 489.235,A -85,B 0,C 180,E1 -11593.302,E2 -11593.302} C_VEL
LIN {X 0,Y 393.327,Z 500.548,A -85,B 0,C 180,E1 -11594.322,E2 -11594.322} C_VEL
LIN {X 0,Y 392.288,Z 510.774,A -85,B 0,C 180,E1 -11595.475,E2 -11595.475} C_VEL
LIN {X 0,Y 391.437,Z 519.976,A -85,B 0,C 180,E1 -11596.768,E2 -11596.768} C_VEL
LIN {X 0,Y 390.457,Z 528.939,A -85,B 0,C 180,E1 -11598.318,E2 -11598.318} C_VEL
LIN {X 0,Y 389.751,Z 536.177,A -85,B 0,C 180,E1 -11599.875,E2 -11599.875} C_VEL
LIN {X 0,Y 389.337,Z 541.083,A -85,B 0,C 180,E1 -11601.175,E2 -11601.175} C_VEL
LIN {X 0,Y 388.975,Z 545.866,A -85,B 0,C 180,E1 -11602.735,E2 -11602.735} C_VEL
LIN {X 0,Y 388.775,Z 548.64,A -85,B 0,C 180,E1 -11603.856,E2 -11603.856} C_VEL
LIN {X 0,Y 388.699,Z 552.221,A -85,B 0,C 180,E1 -11605.854,E2 -11605.854} C_VEL
LIN {X 0,Y 388.659,Z 554.361,A -85,B 0,C 180,E1 -11607.928,E2 -11607.928} C_VEL
LIN {X 0,Y 388.703,Z 554.799,A -85,B 0,C 180,E1 -11608.965,E2 -11608.965} C_VEL
LIN {X 0,Y 388.708,Z 554.844,A -85,B 0,C 180,E1 -11610.001,E2 -11610.001} C_VEL
LIN {X 0,Y 388.704,Z 554.504,A -85,B 0,C 180,E1 -11611.037,E2 -11611.037} C_VEL
LIN {X 0,Y 388.677,Z 553.773,A -85,B 0,C 180,E1 -11612.073,E2 -11612.073} C_VEL
LIN {X 0,Y 388.638,Z 552.597,A -85,B 0,C 180,E1 -11613.111,E2 -11613.111} C_VEL
LIN {X 0,Y 388.713,Z 550.069,A -85,B 0,C 180,E1 -11614.668,E2 -11614.668} C_VEL
LIN {X 0,Y 388.796,Z 546.516,A -85,B 0,C 180,E1 -11616.227,E2 -11616.227} C_VEL
LIN {X 0,Y 388.999,Z 541.843,A -85,B 0,C 180,E1 -11617.789,E2 -11617.789} C_VEL
LIN {X 0,Y 389.44,Z 534.782,A -85,B 0,C 180,E1 -11619.61,E2 -11619.61} C_VEL
LIN {X 0,Y 389.932,Z 527.118,A -85,B 0,C 180,E1 -11621.173,E2 -11621.173} C_VEL
LIN {X 0,Y 390.613,Z 519.272,A -85,B 0,C 180,E1 -11622.47,E2 -11622.47} C_VEL
LIN {X 0,Y 391.493,Z 508.815,A -85,B 0,C 180,E1 -11623.866,E2 -11623.866} C_VEL
LIN {X 0,Y 392.108,Z 498.992,A -85,B 0,C 180,E1 -11624.932,E2 -11624.932} C_VEL
LIN {X 0,Y 393.002,Z 487.042,A -85,B 0,C 180,E1 -11625.96,E2 -11625.96} C_VEL
LIN {X 0,Y 393.791,Z 474.204,A -85,B 0,C 180,E1 -11626.793,E2 -11626.793} C_VEL
LIN {X 0,Y 394.413,Z 462.088,A -85,B 0,C 180,E1 -11627.366,E2 -11627.366} C_VEL
LIN {X 0,Y 394.869,Z 450.135,A -85,B 0,C 180,E1 -11627.747,E2 -11627.747} C_VEL
LIN {X 0,Y 395.791,Z 370.517,A -85,B 0,C 180,E1 -11629.212,E2 -11629.212} C_VEL
LIN {X 0,Y 391.633,Z 342.378,A -85,B 0,C 180,E1 -11629.936,E2 -11629.936} C_VEL
LIN {X 0,Y 392.811,Z 325.664,A -85,B 0,C 180,E1 -11633.459,E2 -11633.459} C_VEL
LIN {X 0,Y 392.876,Z 321.775,A -85,B 0,C 180,E1 -11634.296,E2 -11634.296} C_VEL
LIN {X 0,Y 390.477,Z 308.568,A -85,B 0,C 180,E1 -11637.321,E2 -11637.321} C_VEL
LIN {X 0,Y 390.131,Z 306.891,A -85,B 0,C 180,E1 -11637.747,E2 -11637.747} C_VEL
LIN {X 0,Y 390.028,Z 306.9,A -85,B 0,C 180,E1 -11641.505,E2 -11641.505} C_VEL
LIN {X 0,Y 390.089,Z 306.889,A -85,B 0,C 180,E1 -11645.207,E2 -11645.207} C_VEL
LIN {X 0,Y 390.062,Z 306.893,A -85,B 0,C 180,E1 -11649.097,E2 -11649.097} C_VEL
LIN {X 0,Y 390.041,Z 306.902,A -85,B 0,C 180,E1 -11652.373,E2 -11652.373} C_VEL
LIN {X 0,Y 390.048,Z 306.894,A -85,B 0,C 180,E1 -11655.354,E2 -11655.354} C_VEL
LIN {X 0,Y 390.029,Z 306.9,A -85,B 0,C 180,E1 -11658.186,E2 -11658.186} C_VEL
LIN {X 0,Y 390.087,Z 306.893,A -85,B 0,C 180,E1 -11660.907,E2 -11660.907} C_VEL
LIN {X 0,Y 390.089,Z 306.897,A -85,B 0,C 180,E1 -11664.793,E2 -11664.793} C_VEL
LIN {X 0,Y 390.028,Z 306.9,A -85,B 0,C 180,E1 -11668.496,E2 -11668.496} C_VEL
LIN {X 0,Y 390.079,Z 306.89,A -85,B 0,C 180,E1 -11672.067,E2 -11672.067} C_VEL
LIN {X 0,Y 390.064,Z 306.896,A -85,B 0,C 180,E1 -11675.518,E2 -11675.518} C_VEL
LIN {X 0,Y 390.06,Z 306.895,A -85,B 0,C 180,E1 -11678.878,E2 -11678.878} C_VEL
LIN {X 0,Y 390.116,Z 306.886,A -85,B 0,C 180,E1 -11682.166,E2 -11682.166} C_VEL
LIN {X 0,Y 390.148,Z 306.887,A -85,B 0,C 180,E1 -11685.392,E2 -11685.392} C_VEL
LIN {X 0,Y 390.15,Z 306.882,A -85,B 0,C 180,E1 -11688.571,E2 -11688.571} C_VEL
LIN {X 0,Y 390.274,Z 306.87,A -85,B 0,C 180,E1 -11692.072,E2 -11692.072} C_VEL
LIN {X 0,Y 390.22,Z 306.873,A -85,B 0,C 180,E1 -11694.833,E2 -11694.833} C_VEL
LIN {X 0,Y 390.416,Z 306.855,A -85,B 0,C 180,E1 -11697.937,E2 -11697.937} C_VEL
LIN {X 0,Y 390.547,Z 306.838,A -85,B 0,C 180,E1 -11700,E2 -11700} C_VEL
LIN {X 0,Y 390.28,Z 306.865,A -85,B 0,C 180,E1 -11703.097,E2 -11703.097} C_VEL
LIN {X 0,Y 390.263,Z 306.87,A -85,B 0,C 180,E1 -11706.525,E2 -11706.525} C_VEL
LIN {X 0,Y 390.196,Z 306.876,A -85,B 0,C 180,E1 -11709.329,E2 -11709.329} C_VEL
LIN {X 0,Y 390.174,Z 306.885,A -85,B 0,C 180,E1 -11712.483,E2 -11712.483} C_VEL
LIN {X 0,Y 390.143,Z 306.882,A -85,B 0,C 180,E1 -11715.676,E2 -11715.676} C_VEL
LIN {X 0,Y 390.106,Z 306.894,A -85,B 0,C 180,E1 -11718.922,E2 -11718.922} C_VEL
LIN {X 0,Y 390.04,Z 306.896,A -85,B 0,C 180,E1 -11722.234,E2 -11722.234} C_VEL
LIN {X 0,Y 390.087,Z 306.89,A -85,B 0,C 180,E1 -11725.732,E2 -11725.732} C_VEL
LIN {X 0,Y 390.047,Z 306.901,A -85,B 0,C 180,E1 -11729.11,E2 -11729.11} C_VEL
LIN {X 0,Y 390.045,Z 306.896,A -85,B 0,C 180,E1 -11732.721,E2 -11732.721} C_VEL
LIN {X 0,Y 390.057,Z 306.897,A -85,B 0,C 180,E1 -11735.824,E2 -11735.824} C_VEL
LIN {X 0,Y 390.063,Z 306.895,A -85,B 0,C 180,E1 -11739.216,E2 -11739.216} C_VEL
LIN {X 0,Y 390.041,Z 306.896,A -85,B 0,C 180,E1 -11742.373,E2 -11742.373} C_VEL
LIN {X 0,Y 390.046,Z 306.897,A -85,B 0,C 180,E1 -11745.354,E2 -11745.354} C_VEL
LIN {X 0,Y 390.026,Z 306.902,A -85,B 0,C 180,E1 -11748.185,E2 -11748.185} C_VEL
LIN {X 0,Y 390.067,Z 306.892,A -85,B 0,C 180,E1 -11750.904,E2 -11750.904} C_VEL
LIN {X 0,Y 390.086,Z 306.891,A -85,B 0,C 180,E1 -11754.792,E2 -11754.792} C_VEL
LIN {X 0,Y 390.025,Z 306.903,A -85,B 0,C 180,E1 -11758.495,E2 -11758.495} C_VEL
LIN {X 0,Y 390.076,Z 306.893,A -85,B 0,C 180,E1 -11762.066,E2 -11762.066} C_VEL
LIN {X 0,Y 390.064,Z 306.892,A -85,B 0,C 180,E1 -11765.517,E2 -11765.517} C_VEL
LIN {X 0,Y 390.057,Z 306.899,A -85,B 0,C 180,E1 -11768.877,E2 -11768.877} C_VEL
LIN {X 0,Y 390.112,Z 306.887,A -85,B 0,C 180,E1 -11772.165,E2 -11772.165} C_VEL
LIN {X 0,Y 390.144,Z 306.885,A -85,B 0,C 180,E1 -11775.392,E2 -11775.392} C_VEL
LIN {X 0,Y 390.146,Z 306.884,A -85,B 0,C 180,E1 -11778.57,E2 -11778.57} C_VEL
LIN {X 0,Y 390.206,Z 306.996,A -85,B 0,C 180,E1 -11780.507,E2 -11780.507} C_VEL
LIN {X 0,Y 391.89,Z 316.205,A -85,B 0,C 180,E1 -11782.787,E2 -11782.787} C_VEL
LIN {X 0,Y 391.836,Z 322.163,A -85,B 0,C 180,E1 -11784.161,E2 -11784.161} C_VEL
LIN {X 0,Y 396.145,Z 345.606,A -85,B 0,C 180,E1 -11784.791,E2 -11784.791} C_VEL
LIN {X 0,Y 394.957,Z 429.785,A -85,B 0,C 180,E1 -11786.341,E2 -11786.341} C_VEL
LIN {X 0,Y 394.536,Z 442.284,A -85,B 0,C 180,E1 -11786.761,E2 -11786.761} C_VEL
LIN {X 0,Y 394.068,Z 453.93,A -85,B 0,C 180,E1 -11787.337,E2 -11787.337} C_VEL
LIN {X 0,Y 393.414,Z 465.238,A -85,B 0,C 180,E1 -11788.08,E2 -11788.08} C_VEL
LIN {X 0,Y 392.688,Z 475.881,A -85,B 0,C 180,E1 -11788.974,E2 -11788.974} C_VEL
LIN {X 0,Y 391.863,Z 486.747,A -85,B 0,C 180,E1 -11790.128,E2 -11790.128} C_VEL
LIN {X 0,Y 391.131,Z 495.618,A -85,B 0,C 180,E1 -11791.286,E2 -11791.286} C_VEL
LIN {X 0,Y 390.323,Z 505.257,A -85,B 0,C 180,E1 -11792.837,E2 -11792.837} C_VEL
LIN {X 0,Y 389.75,Z 512.92,A -85,B 0,C 180,E1 -11794.394,E2 -11794.394} C_VEL
LIN {X 0,Y 389.417,Z 518.168,A -85,B 0,C 180,E1 -11795.696,E2 -11795.696} C_VEL
LIN {X 0,Y 389.118,Z 523.253,A -85,B 0,C 180,E1 -11797.262,E2 -11797.262} C_VEL
LIN {X 0,Y 388.984,Z 525.301,A -85,B 0,C 180,E1 -11798.031,E2 -11798.031} C_VEL
LIN {X 0,Y 388.171,Z 527.257,A -85,B 0,C 180,E1 -11798.847,E2 -11798.847} C_VEL
LIN {X 0,Y 385.132,Z 529.88,A -85,B 0,C 180,E1 -11800.191,E2 -11800.191} C_VEL
LIN {X 0,Y 382.646,Z 531.467,A -85,B 0,C 180,E1 -11801.297,E2 -11801.297} C_VEL
LIN {X 0,Y 381.605,Z 532.36,A -85,B 0,C 180,E1 -11802.162,E2 -11802.162} C_VEL
LIN {X 0,Y 381.531,Z 532.58,A -85,B 0,C 180,E1 -11802.455,E2 -11802.455} C_VEL
LIN {X 0,Y 381.445,Z 533.287,A -85,B 0,C 180,E1 -11803.857,E2 -11803.857} C_VEL
LIN {X 0,Y 381.413,Z 533.335,A -85,B 0,C 180,E1 -11804.948,E2 -11804.948} C_VEL
LIN {X 0,Y 381.536,Z 532.551,A -85,B 0,C 180,E1 -11806.694,E2 -11806.694} C_VEL
LIN {X 0,Y 381.68,Z 530.953,A -85,B 0,C 180,E1 -11808.241,E2 -11808.241} C_VEL
LIN {X 0,Y 382.046,Z 527.551,A -85,B 0,C 180,E1 -11810.252,E2 -11810.252} C_VEL
LIN {X 0,Y 382.484,Z 522.917,A -85,B 0,C 180,E1 -11812.127,E2 -11812.127} C_VEL
LIN {X 0,Y 383.089,Z 517.401,A -85,B 0,C 180,E1 -11813.802,E2 -11813.802} C_VEL
LIN {X 0,Y 383.903,Z 510.395,A -85,B 0,C 180,E1 -11815.479,E2 -11815.479} C_VEL
LIN {X 0,Y 384.729,Z 503.016,A -85,B 0,C 180,E1 -11816.905,E2 -11816.905} C_VEL
LIN {X 0,Y 385.659,Z 494.336,A -85,B 0,C 180,E1 -11818.28,E2 -11818.28} C_VEL
LIN {X 0,Y 386.746,Z 484.52,A -85,B 0,C 180,E1 -11819.531,E2 -11819.531} C_VEL
LIN {X 0,Y 387.822,Z 473.692,A -85,B 0,C 180,E1 -11820.641,E2 -11820.641} C_VEL
LIN {X 0,Y 388.807,Z 461.664,A -85,B 0,C 180,E1 -11821.613,E2 -11821.613} C_VEL
LIN {X 0,Y 389.66,Z 449.151,A -85,B 0,C 180,E1 -11822.363,E2 -11822.363} C_VEL
LIN {X 0,Y 390.266,Z 436.814,A -85,B 0,C 180,E1 -11822.891,E2 -11822.891} C_VEL
LIN {X 0,Y 390.662,Z 423.911,A -85,B 0,C 180,E1 -11823.238,E2 -11823.238} C_VEL
LIN {X 0,Y 392.012,Z 346.728,A -85,B 0,C 180,E1 -11824.679,E2 -11824.679} C_VEL
LIN {X 0,Y 387.859,Z 328.182,A -85,B 0,C 180,E1 -11825.329,E2 -11825.329} C_VEL
LIN {X 0,Y 386.115,Z 322.259,A -85,B 0,C 180,E1 -11825.584,E2 -11825.584} C_VEL
LIN {X 0,Y 383.744,Z 311.021,A -85,B 0,C 180,E1 -11828.511,E2 -11828.511} C_VEL
LIN {X 0,Y 382.976,Z 307.779,A -85,B 0,C 180,E1 -11829.427,E2 -11829.427} C_VEL
LIN {X 0,Y 382.999,Z 307.78,A -85,B 0,C 180,E1 -11832.778,E2 -11832.778} C_VEL
LIN {X 0,Y 382.988,Z 307.778,A -85,B 0,C 180,E1 -11835.788,E2 -11835.788} C_VEL
LIN {X 0,Y 382.954,Z 307.782,A -85,B 0,C 180,E1 -11838.8,E2 -11838.8} C_VEL
LIN {X 0,Y 382.986,Z 307.775,A -85,B 0,C 180,E1 -11842.097,E2 -11842.097} C_VEL
LIN {X 0,Y 383.008,Z 307.763,A -85,B 0,C 180,E1 -11845.331,E2 -11845.331} C_VEL
LIN {X 0,Y 382.973,Z 307.781,A -85,B 0,C 180,E1 -11849.081,E2 -11849.081} C_VEL
LIN {X 0,Y 382.982,Z 307.777,A -85,B 0,C 180,E1 -11852.693,E2 -11852.693} C_VEL
LIN {X 0,Y 383.001,Z 307.775,A -85,B 0,C 180,E1 -11856.191,E2 -11856.191} C_VEL
LIN {X 0,Y 383.047,Z 307.771,A -85,B 0,C 180,E1 -11859.598,E2 -11859.598} C_VEL
LIN {X 0,Y 383.06,Z 307.763,A -85,B 0,C 180,E1 -11862.93,E2 -11862.93} C_VEL
LIN {X 0,Y 383.116,Z 307.753,A -85,B 0,C 180,E1 -11866.464,E2 -11866.464} C_VEL
LIN {X 0,Y 383.126,Z 307.753,A -85,B 0,C 180,E1 -11870.498,E2 -11870.498} C_VEL
LIN {X 0,Y 383.219,Z 307.746,A -85,B 0,C 180,E1 -11873.683,E2 -11873.683} C_VEL
LIN {X 0,Y 383.356,Z 307.724,A -85,B 0,C 180,E1 -11877.899,E2 -11877.899} C_VEL
LIN {X 0,Y 383.358,Z 307.723,A -85,B 0,C 180,E1 -11882.101,E2 -11882.101} C_VEL
LIN {X 0,Y 383.25,Z 307.745,A -85,B 0,C 180,E1 -11886.317,E2 -11886.317} C_VEL
LIN {X 0,Y 383.13,Z 307.755,A -85,B 0,C 180,E1 -11889.503,E2 -11889.503} C_VEL
LIN {X 0,Y 383.117,Z 307.751,A -85,B 0,C 180,E1 -11893.537,E2 -11893.537} C_VEL
LIN {X 0,Y 383.086,Z 307.759,A -85,B 0,C 180,E1 -11897.07,E2 -11897.07} C_VEL
LIN {X 0,Y 383.021,Z 307.771,A -85,B 0,C 180,E1 -11900.647,E2 -11900.647} C_VEL
LIN {X 0,Y 383.002,Z 307.771,A -85,B 0,C 180,E1 -11903.81,E2 -11903.81} C_VEL
LIN {X 0,Y 382.984,Z 307.773,A -85,B 0,C 180,E1 -11907.308,E2 -11907.308} C_VEL
LIN {X 0,Y 382.975,Z 307.779,A -85,B 0,C 180,E1 -11910.92,E2 -11910.92} C_VEL
LIN {X 0,Y 383.012,Z 307.772,A -85,B 0,C 180,E1 -11914.669,E2 -11914.669} C_VEL
LIN {X 0,Y 382.988,Z 307.776,A -85,B 0,C 180,E1 -11917.903,E2 -11917.903} C_VEL
LIN {X 0,Y 382.958,Z 307.784,A -85,B 0,C 180,E1 -11921.351,E2 -11921.351} C_VEL
LIN {X 0,Y 382.99,Z 307.768,A -85,B 0,C 180,E1 -11924.304,E2 -11924.304} C_VEL
LIN {X 0,Y 383.006,Z 307.778,A -85,B 0,C 180,E1 -11927.241,E2 -11927.241} C_VEL
LIN {X 0,Y 383.006,Z 307.78,A -85,B 0,C 180,E1 -11930.416,E2 -11930.416} C_VEL
LIN {X 0,Y 383.021,Z 307.777,A -85,B 0,C 180,E1 -11934.046,E2 -11934.046} C_VEL
LIN {X 0,Y 382.984,Z 307.777,A -85,B 0,C 180,E1 -11937.579,E2 -11937.579} C_VEL
LIN {X 0,Y 383.063,Z 307.944,A -85,B 0,C 180,E1 -11940.391,E2 -11940.391} C_VEL
LIN {X 0,Y 385.287,Z 317.533,A -85,B 0,C 180,E1 -11942.87,E2 -11942.87} C_VEL
LIN {X 0,Y 387.108,Z 327.502,A -85,B 0,C 180,E1 -11945.32,E2 -11945.32} C_VEL
LIN {X 0,Y 386.397,Z 336.278,A -85,B 0,C 180,E1 -11947.264,E2 -11947.264} C_VEL
LIN {X 0,Y 385.914,Z 342,A -85,B 0,C 180,E1 -11948.477,E2 -11948.477} C_VEL
LIN {X 0,Y 390.21,Z 363.626,A -85,B 0,C 180,E1 -11949.199,E2 -11949.199} C_VEL
LIN {X 0,Y 391.649,Z 373.43,A -85,B 0,C 180,E1 -11949.487,E2 -11949.487} C_VEL
LIN {X 0,Y 390.361,Z 450.659,A -85,B 0,C 180,E1 -11950.961,E2 -11950.961} C_VEL
LIN {X 0,Y 389.583,Z 464.292,A -85,B 0,C 180,E1 -11951.428,E2 -11951.428} C_VEL
LIN {X 0,Y 388.741,Z 477.198,A -85,B 0,C 180,E1 -11952.102,E2 -11952.102} C_VEL
LIN {X 0,Y 387.631,Z 489.723,A -85,B 0,C 180,E1 -11953.002,E2 -11953.002} C_VEL
LIN {X 0,Y 386.513,Z 500.901,A -85,B 0,C 180,E1 -11954.038,E2 -11954.038} C_VEL
LIN {X 0,Y 385.432,Z 510.999,A -85,B 0,C 180,E1 -11955.211,E2 -11955.211} C_VEL
LIN {X 0,Y 384.521,Z 520.118,A -85,B 0,C 180,E1 -11956.525,E2 -11956.525} C_VEL
LIN {X 0,Y 383.494,Z 529.024,A -85,B 0,C 180,E1 -11958.103,E2 -11958.103} C_VEL
LIN {X 0,Y 382.741,Z 536.212,A -85,B 0,C 180,E1 -11959.688,E2 -11959.688} C_VEL
LIN {X 0,Y 382.147,Z 542.781,A -85,B 0,C 180,E1 -11961.541,E2 -11961.541} C_VEL
LIN {X 0,Y 381.802,Z 547.143,A -85,B 0,C 180,E1 -11963.129,E2 -11963.129} C_VEL
LIN {X 0,Y 381.645,Z 550.447,A -85,B 0,C 180,E1 -11964.718,E2 -11964.718} C_VEL
LIN {X 0,Y 381.625,Z 552.098,A -85,B 0,C 180,E1 -11965.777,E2 -11965.777} C_VEL
LIN {X 0,Y 381.545,Z 553.349,A -85,B 0,C 180,E1 -11966.833,E2 -11966.833} C_VEL
LIN {X 0,Y 381.558,Z 554.192,A -85,B 0,C 180,E1 -11967.89,E2 -11967.89} C_VEL
LIN {X 0,Y 381.603,Z 554.608,A -85,B 0,C 180,E1 -11968.946,E2 -11968.946} C_VEL
LIN {X 0,Y 381.639,Z 554.638,A -85,B 0,C 180,E1 -11970.001,E2 -11970.001} C_VEL
LIN {X 0,Y 381.619,Z 554.281,A -85,B 0,C 180,E1 -11971.056,E2 -11971.056} C_VEL
LIN {X 0,Y 381.576,Z 553.525,A -85,B 0,C 180,E1 -11972.112,E2 -11972.112} C_VEL
LIN {X 0,Y 381.627,Z 550.716,A -85,B 0,C 180,E1 -11974.225,E2 -11974.225} C_VEL
LIN {X 0,Y 381.688,Z 546.746,A -85,B 0,C 180,E1 -11976.119,E2 -11976.119} C_VEL
LIN {X 0,Y 381.926,Z 541.451,A -85,B 0,C 180,E1 -11977.934,E2 -11977.934} C_VEL
LIN {X 0,Y 382.39,Z 534.34,A -85,B 0,C 180,E1 -11979.789,E2 -11979.789} C_VEL
LIN {X 0,Y 382.93,Z 526.611,A -85,B 0,C 180,E1 -11981.38,E2 -11981.38} C_VEL
LIN {X 0,Y 383.622,Z 518.688,A -85,B 0,C 180,E1 -11982.701,E2 -11982.701} C_VEL
LIN {X 0,Y 384.509,Z 508.657,A -85,B 0,C 180,E1 -11984.06,E2 -11984.06} C_VEL
LIN {X 0,Y 385.207,Z 498.231,A -85,B 0,C 180,E1 -11985.206,E2 -11985.206} C_VEL
LIN {X 0,Y 386.015,Z 487.812,A -85,B 0,C 180,E1 -11986.121,E2 -11986.121} C_VEL
LIN {X 0,Y 386.856,Z 475.303,A -85,B 0,C 180,E1 -11986.967,E2 -11986.967} C_VEL
LIN {X 0,Y 387.5,Z 462.864,A -85,B 0,C 180,E1 -11987.584,E2 -11987.584} C_VEL
LIN {X 0,Y 388.015,Z 450.279,A -85,B 0,C 180,E1 -11988.003,E2 -11988.003} C_VEL
LIN {X 0,Y 388.976,Z 371.332,A -85,B 0,C 180,E1 -11989.484,E2 -11989.484} C_VEL
LIN {X 0,Y 384.706,Z 342.249,A -85,B 0,C 180,E1 -11990.232,E2 -11990.232} C_VEL
LIN {X 0,Y 385.842,Z 326.448,A -85,B 0,C 180,E1 -11993.624,E2 -11993.624} C_VEL
LIN {X 0,Y 385.893,Z 322.872,A -85,B 0,C 180,E1 -11994.409,E2 -11994.409} C_VEL
LIN {X 0,Y 383.413,Z 309.346,A -85,B 0,C 180,E1 -11997.569,E2 -11997.569} C_VEL
LIN {X 0,Y 383.086,Z 307.769,A -85,B 0,C 180,E1 -11997.958,E2 -11997.958} C_VEL
LIN {X 0,Y 382.988,Z 307.774,A -85,B 0,C 180,E1 -12000.919,E2 -12000.919} C_VEL
LIN {X 0,Y 383.022,Z 307.77,A -85,B 0,C 180,E1 -12004.668,E2 -12004.668} C_VEL
LIN {X 0,Y 382.998,Z 307.777,A -85,B 0,C 180,E1 -12007.903,E2 -12007.903} C_VEL
LIN {X 0,Y 382.967,Z 307.776,A -85,B 0,C 180,E1 -12011.351,E2 -12011.351} C_VEL
LIN {X 0,Y 383,Z 307.779,A -85,B 0,C 180,E1 -12014.303,E2 -12014.303} C_VEL
LIN {X 0,Y 383.015,Z 307.771,A -85,B 0,C 180,E1 -12017.24,E2 -12017.24} C_VEL
LIN {X 0,Y 383.009,Z 307.776,A -85,B 0,C 180,E1 -12020.416,E2 -12020.416} C_VEL
LIN {X 0,Y 383.029,Z 307.769,A -85,B 0,C 180,E1 -12024.044,E2 -12024.044} C_VEL
LIN {X 0,Y 382.991,Z 307.774,A -85,B 0,C 180,E1 -12027.578,E2 -12027.578} C_VEL
LIN {X 0,Y 382.989,Z 307.775,A -85,B 0,C 180,E1 -12030.3,E2 -12030.3} C_VEL
LIN {X 0,Y 383.047,Z 307.766,A -85,B 0,C 180,E1 -12034.033,E2 -12034.033} C_VEL
LIN {X 0,Y 382.996,Z 307.779,A -85,B 0,C 180,E1 -12037.334,E2 -12037.334} C_VEL
LIN {X 0,Y 383.063,Z 307.765,A -85,B 0,C 180,E1 -12040.716,E2 -12040.716} C_VEL
LIN {X 0,Y 383.085,Z 307.763,A -85,B 0,C 180,E1 -12044.027,E2 -12044.027} C_VEL
LIN {X 0,Y 383.14,Z 307.758,A -85,B 0,C 180,E1 -12047.284,E2 -12047.284} C_VEL
LIN {X 0,Y 383.146,Z 307.755,A -85,B 0,C 180,E1 -12050.498,E2 -12050.498} C_VEL
LIN {X 0,Y 383.273,Z 307.743,A -85,B 0,C 180,E1 -12053.683,E2 -12053.683} C_VEL
LIN {X 0,Y 383.382,Z 307.731,A -85,B 0,C 180,E1 -12057.899,E2 -12057.899} C_VEL
LIN {X 0,Y 383.517,Z 307.714,A -85,B 0,C 180,E1 -12060,E2 -12060} C_VEL
LIN {X 0,Y 383.218,Z 307.745,A -85,B 0,C 180,E1 -12063.154,E2 -12063.154} C_VEL
LIN {X 0,Y 383.228,Z 307.749,A -85,B 0,C 180,E1 -12066.513,E2 -12066.513} C_VEL
LIN {X 0,Y 383.147,Z 307.754,A -85,B 0,C 180,E1 -12069.502,E2 -12069.502} C_VEL
LIN {X 0,Y 383.129,Z 307.756,A -85,B 0,C 180,E1 -12073.536,E2 -12073.536} C_VEL
LIN {X 0,Y 383.097,Z 307.764,A -85,B 0,C 180,E1 -12077.069,E2 -12077.069} C_VEL
LIN {X 0,Y 383.032,Z 307.773,A -85,B 0,C 180,E1 -12080.646,E2 -12080.646} C_VEL
LIN {X 0,Y 383.02,Z 307.77,A -85,B 0,C 180,E1 -12083.808,E2 -12083.808} C_VEL
LIN {X 0,Y 383.021,Z 307.775,A -85,B 0,C 180,E1 -12087.304,E2 -12087.304} C_VEL
LIN {X 0,Y 382.985,Z 307.777,A -85,B 0,C 180,E1 -12090.918,E2 -12090.918} C_VEL
LIN {X 0,Y 383.02,Z 307.77,A -85,B 0,C 180,E1 -12094.667,E2 -12094.667} C_VEL
LIN {X 0,Y 382.999,Z 307.776,A -85,B 0,C 180,E1 -12097.903,E2 -12097.903} C_VEL
LIN {X 0,Y 382.972,Z 307.779,A -85,B 0,C 180,E1 -12101.349,E2 -12101.349} C_VEL
LIN {X 0,Y 382.997,Z 307.775,A -85,B 0,C 180,E1 -12104.303,E2 -12104.303} C_VEL
LIN {X 0,Y 383.012,Z 307.772,A -85,B 0,C 180,E1 -12107.24,E2 -12107.24} C_VEL
LIN {X 0,Y 382.996,Z 307.776,A -85,B 0,C 180,E1 -12110.417,E2 -12110.417} C_VEL
LIN {X 0,Y 383.026,Z 307.775,A -85,B 0,C 180,E1 -12114.044,E2 -12114.044} C_VEL
LIN {X 0,Y 382.989,Z 307.774,A -85,B 0,C 180,E1 -12117.577,E2 -12117.577} C_VEL
LIN {X 0,Y 382.986,Z 307.78,A -85,B 0,C 180,E1 -12120.299,E2 -12120.299} C_VEL
LIN {X 0,Y 383.044,Z 307.769,A -85,B 0,C 180,E1 -12124.032,E2 -12124.032} C_VEL
LIN {X 0,Y 382.998,Z 307.774,A -85,B 0,C 180,E1 -12127.334,E2 -12127.334} C_VEL
LIN {X 0,Y 383.059,Z 307.771,A -85,B 0,C 180,E1 -12130.715,E2 -12130.715} C_VEL
LIN {X 0,Y 383.081,Z 307.762,A -85,B 0,C 180,E1 -12134.026,E2 -12134.026} C_VEL
LIN {X 0,Y 383.137,Z 307.76,A -85,B 0,C 180,E1 -12137.283,E2 -12137.283} C_VEL
LIN {X 0,Y 383.181,Z 307.876,A -85,B 0,C 180,E1 -12140.298,E2 -12140.298} C_VEL
LIN {X 0,Y 385.008,Z 318.325,A -85,B 0,C 180,E1 -12142.921,E2 -12142.921} C_VEL
LIN {X 0,Y 384.899,Z 322.475,A -85,B 0,C 180,E1 -12143.853,E2 -12143.853} C_VEL
LIN {X 0,Y 389.332,Z 345.995,A -85,B 0,C 180,E1 -12144.503,E2 -12144.503} C_VEL
LIN {X 0,Y 388.127,Z 429.752,A -85,B 0,C 180,E1 -12146.071,E2 -12146.071} C_VEL
LIN {X 0,Y 387.669,Z 442.136,A -85,B 0,C 180,E1 -12146.489,E2 -12146.489} C_VEL
LIN {X 0,Y 387.173,Z 454.511,A -85,B 0,C 180,E1 -12147.112,E2 -12147.112} C_VEL
LIN {X 0,Y 386.441,Z 466.375,A -85,B 0,C 180,E1 -12147.915,E2 -12147.915} C_VEL
LIN {X 0,Y 385.624,Z 478.074,A -85,B 0,C 180,E1 -12148.955,E2 -12148.955} C_VEL
LIN {X 0,Y 384.772,Z 488.586,A -85,B 0,C 180,E1 -12150.13,E2 -12150.13} C_VEL
LIN {X 0,Y 384.039,Z 497.183,A -85,B 0,C 180,E1 -12151.31,E2 -12151.31} C_VEL
LIN {X 0,Y 383.342,Z 505.112,A -85,B 0,C 180,E1 -12152.626,E2 -12152.626} C_VEL
LIN {X 0,Y 382.728,Z 512.859,A -85,B 0,C 180,E1 -12154.211,E2 -12154.211} C_VEL
LIN {X 0,Y 382.328,Z 519.063,A -85,B 0,C 180,E1 -12155.802,E2 -12155.802} C_VEL
LIN {X 0,Y 382.021,Z 524.003,A -85,B 0,C 180,E1 -12157.398,E2 -12157.398} C_VEL
LIN {X 0,Y 381.742,Z 527.823,A -85,B 0,C 180,E1 -12159.002,E2 -12159.002} C_VEL
LIN {X 0,Y 381.566,Z 530.606,A -85,B 0,C 180,E1 -12160.613,E2 -12160.613} C_VEL
LIN {X 0,Y 381.531,Z 532.58,A -85,B 0,C 180,E1 -12162.455,E2 -12162.455} C_VEL
LIN {X 0,Y 380.873,Z 533.193,A -85,B 0,C 180,E1 -12163.331,E2 -12163.331} C_VEL
LIN {X 0,Y 377.969,Z 533.556,A -85,B 0,C 180,E1 -12164.762,E2 -12164.762} C_VEL
LIN {X 0,Y 375.533,Z 533.271,A -85,B 0,C 180,E1 -12165.919,E2 -12165.919} C_VEL
LIN {X 0,Y 374.535,Z 532.741,A -85,B 0,C 180,E1 -12166.812,E2 -12166.812} C_VEL
LIN {X 0,Y 374.481,Z 532.488,A -85,B 0,C 180,E1 -12167.113,E2 -12167.113} C_VEL
LIN {X 0,Y 374.654,Z 530.864,A -85,B 0,C 180,E1 -12168.595,E2 -12168.595} C_VEL
LIN {X 0,Y 374.993,Z 527.743,A -85,B 0,C 180,E1 -12170.433,E2 -12170.433} C_VEL
LIN {X 0,Y 375.388,Z 524.069,A -85,B 0,C 180,E1 -12171.988,E2 -12171.988} C_VEL
LIN {X 0,Y 376.08,Z 518.162,A -85,B 0,C 180,E1 -12173.894,E2 -12173.894} C_VEL
LIN {X 0,Y 376.945,Z 510.904,A -85,B 0,C 180,E1 -12175.688,E2 -12175.688} C_VEL
LIN {X 0,Y 377.79,Z 504.056,A -85,B 0,C 180,E1 -12177.053,E2 -12177.053} C_VEL
LIN {X 0,Y 378.801,Z 495.003,A -85,B 0,C 180,E1 -12178.537,E2 -12178.537} C_VEL
LIN {X 0,Y 379.909,Z 485.806,A -85,B 0,C 180,E1 -12179.752,E2 -12179.752} C_VEL
LIN {X 0,Y 381.074,Z 474.637,A -85,B 0,C 180,E1 -12180.935,E2 -12180.935} C_VEL
LIN {X 0,Y 382.11,Z 462.807,A -85,B 0,C 180,E1 -12181.922,E2 -12181.922} C_VEL
LIN {X 0,Y 383.026,Z 450.265,A -85,B 0,C 180,E1 -12182.707,E2 -12182.707} C_VEL
LIN {X 0,Y 383.704,Z 437.101,A -85,B 0,C 180,E1 -12183.287,E2 -12183.287} C_VEL
LIN {X 0,Y 384.134,Z 424.115,A -85,B 0,C 180,E1 -12183.642,E2 -12183.642} C_VEL
LIN {X 0,Y 385.547,Z 347.89,A -85,B 0,C 180,E1 -12185.088,E2 -12185.088} C_VEL
LIN {X 0,Y 381.656,Z 330.457,A -85,B 0,C 180,E1 -12185.716,E2 -12185.716} C_VEL
LIN {X 0,Y 379.916,Z 325.053,A -85,B 0,C 180,E1 -12185.954,E2 -12185.954} C_VEL
LIN {X 0,Y 378.945,Z 322.458,A -85,B 0,C 180,E1 -12186.1,E2 -12186.1} C_VEL
LIN {X 0,Y 376.608,Z 311.438,A -85,B 0,C 180,E1 -12189.039,E2 -12189.039} C_VEL
LIN {X 0,Y 375.926,Z 308.657,A -85,B 0,C 180,E1 -12189.813,E2 -12189.813} C_VEL
LIN {X 0,Y 375.927,Z 308.66,A -85,B 0,C 180,E1 -12193.189,E2 -12193.189} C_VEL
LIN {X 0,Y 375.926,Z 308.652,A -85,B 0,C 180,E1 -12196.81,E2 -12196.81} C_VEL
LIN {X 0,Y 375.928,Z 308.656,A -85,B 0,C 180,E1 -12200.533,E2 -12200.533} C_VEL
LIN {X 0,Y 375.954,Z 308.658,A -85,B 0,C 180,E1 -12203.495,E2 -12203.495} C_VEL
LIN {X 0,Y 375.95,Z 308.637,A -85,B 0,C 180,E1 -12205.888,E2 -12205.888} C_VEL
LIN {X 0,Y 375.953,Z 308.654,A -85,B 0,C 180,E1 -12209.687,E2 -12209.687} C_VEL
LIN {X 0,Y 375.925,Z 308.658,A -85,B 0,C 180,E1 -12212.136,E2 -12212.136} C_VEL
LIN {X 0,Y 375.95,Z 308.657,A -85,B 0,C 180,E1 -12215.716,E2 -12215.716} C_VEL
LIN {X 0,Y 375.971,Z 308.648,A -85,B 0,C 180,E1 -12219.197,E2 -12219.197} C_VEL
LIN {X 0,Y 376,Z 308.643,A -85,B 0,C 180,E1 -12222.599,E2 -12222.599} C_VEL
LIN {X 0,Y 376.08,Z 308.629,A -85,B 0,C 180,E1 -12226.343,E2 -12226.343} C_VEL
LIN {X 0,Y 376.097,Z 308.63,A -85,B 0,C 180,E1 -12230.318,E2 -12230.318} C_VEL
LIN {X 0,Y 376.18,Z 308.622,A -85,B 0,C 180,E1 -12233.564,E2 -12233.564} C_VEL
LIN {X 0,Y 376.32,Z 308.6,A -85,B 0,C 180,E1 -12237.86,E2 -12237.86} C_VEL
LIN {X 0,Y 376.322,Z 308.599,A -85,B 0,C 180,E1 -12242.141,E2 -12242.141} C_VEL
LIN {X 0,Y 376.209,Z 308.619,A -85,B 0,C 180,E1 -12246.436,E2 -12246.436} C_VEL
LIN {X 0,Y 376.101,Z 308.631,A -85,B 0,C 180,E1 -12249.682,E2 -12249.682} C_VEL
LIN {X 0,Y 376.081,Z 308.627,A -85,B 0,C 180,E1 -12253.658,E2 -12253.658} C_VEL
LIN {X 0,Y 376.024,Z 308.635,A -85,B 0,C 180,E1 -12257.401,E2 -12257.401} C_VEL
LIN {X 0,Y 375.971,Z 308.651,A -85,B 0,C 180,E1 -12260.833,E2 -12260.833} C_VEL
LIN {X 0,Y 375.928,Z 308.651,A -85,B 0,C 180,E1 -12264.286,E2 -12264.286} C_VEL
LIN {X 0,Y 375.919,Z 308.656,A -85,B 0,C 180,E1 -12266.66,E2 -12266.66} C_VEL
LIN {X 0,Y 375.912,Z 308.657,A -85,B 0,C 180,E1 -12269.084,E2 -12269.084} C_VEL
LIN {X 0,Y 375.951,Z 308.65,A -85,B 0,C 180,E1 -12271.563,E2 -12271.563} C_VEL
LIN {X 0,Y 375.951,Z 308.651,A -85,B 0,C 180,E1 -12275.417,E2 -12275.417} C_VEL
LIN {X 0,Y 375.93,Z 308.653,A -85,B 0,C 180,E1 -12278.264,E2 -12278.264} C_VEL
LIN {X 0,Y 375.914,Z 308.657,A -85,B 0,C 180,E1 -12281.599,E2 -12281.599} C_VEL
LIN {X 0,Y 375.921,Z 308.655,A -85,B 0,C 180,E1 -12284.732,E2 -12284.732} C_VEL
LIN {X 0,Y 375.928,Z 308.662,A -85,B 0,C 180,E1 -12288.401,E2 -12288.401} C_VEL
LIN {X 0,Y 375.967,Z 308.655,A -85,B 0,C 180,E1 -12291.731,E2 -12291.731} C_VEL
LIN {X 0,Y 375.977,Z 308.646,A -85,B 0,C 180,E1 -12295.334,E2 -12295.334} C_VEL
LIN {X 0,Y 375.956,Z 308.653,A -85,B 0,C 180,E1 -12298.439,E2 -12298.439} C_VEL
LIN {X 0,Y 375.995,Z 308.699,A -85,B 0,C 180,E1 -12299.924,E2 -12299.924} C_VEL
LIN {X 0,Y 378.51,Z 319.571,A -85,B 0,C 180,E1 -12302.801,E2 -12302.801} C_VEL
LIN {X 0,Y 380.241,Z 329.005,A -85,B 0,C 180,E1 -12305.164,E2 -12305.164} C_VEL
LIN {X 0,Y 379.417,Z 338.688,A -85,B 0,C 180,E1 -12307.348,E2 -12307.348} C_VEL
LIN {X 0,Y 379.108,Z 341.565,A -85,B 0,C 180,E1 -12307.987,E2 -12307.987} C_VEL
LIN {X 0,Y 383.542,Z 363.48,A -85,B 0,C 180,E1 -12308.752,E2 -12308.752} C_VEL
LIN {X 0,Y 385.122,Z 374.406,A -85,B 0,C 180,E1 -12309.08,E2 -12309.08} C_VEL
LIN {X 0,Y 383.812,Z 450.202,A -85,B 0,C 180,E1 -12310.55,E2 -12310.55} C_VEL
LIN {X 0,Y 383.08,Z 463.239,A -85,B 0,C 180,E1 -12310.997,E2 -12310.997} C_VEL
LIN {X 0,Y 382.217,Z 475.853,A -85,B 0,C 180,E1 -12311.647,E2 -12311.647} C_VEL
LIN {X 0,Y 381.182,Z 487.111,A -85,B 0,C 180,E1 -12312.429,E2 -12312.429} C_VEL
LIN {X 0,Y 380.011,Z 498.733,A -85,B 0,C 180,E1 -12313.481,E2 -12313.481} C_VEL
LIN {X 0,Y 378.746,Z 509.604,A -85,B 0,C 180,E1 -12314.721,E2 -12314.721} C_VEL
LIN {X 0,Y 377.812,Z 518.65,A -85,B 0,C 180,E1 -12316.007,E2 -12316.007} C_VEL
LIN {X 0,Y 376.881,Z 526.415,A -85,B 0,C 180,E1 -12317.344,E2 -12317.344} C_VEL
LIN {X 0,Y 375.99,Z 534.022,A -85,B 0,C 180,E1 -12318.955,E2 -12318.955} C_VEL
LIN {X 0,Y 375.253,Z 541.066,A -85,B 0,C 180,E1 -12320.841,E2 -12320.841} C_VEL
LIN {X 0,Y 374.868,Z 545.767,A -85,B 0,C 180,E1 -12322.46,E2 -12322.46} C_VEL
LIN {X 0,Y 374.59,Z 549.063,A -85,B 0,C 180,E1 -12323.924,E2 -12323.924} C_VEL
LIN {X 0,Y 374.529,Z 551.975,A -85,B 0,C 180,E1 -12325.696,E2 -12325.696} C_VEL
LIN {X 0,Y 374.46,Z 553.209,A -85,B 0,C 180,E1 -12326.773,E2 -12326.773} C_VEL
LIN {X 0,Y 374.456,Z 554.018,A -85,B 0,C 180,E1 -12327.85,E2 -12327.85} C_VEL
LIN {X 0,Y 374.503,Z 554.417,A -85,B 0,C 180,E1 -12328.926,E2 -12328.926} C_VEL
LIN {X 0,Y 374.554,Z 554.43,A -85,B 0,C 180,E1 -12330.001,E2 -12330.001} C_VEL
LIN {X 0,Y 374.52,Z 554.056,A -85,B 0,C 180,E1 -12331.076,E2 -12331.076} C_VEL
LIN {X 0,Y 374.475,Z 553.269,A -85,B 0,C 180,E1 -12332.152,E2 -12332.152} C_VEL
LIN {X 0,Y 374.555,Z 550.422,A -85,B 0,C 180,E1 -12334.305,E2 -12334.305} C_VEL
LIN {X 0,Y 374.584,Z 546.802,A -85,B 0,C 180,E1 -12336.068,E2 -12336.068} C_VEL
LIN {X 0,Y 374.774,Z 542.769,A -85,B 0,C 180,E1 -12337.544,E2 -12337.544} C_VEL
LIN {X 0,Y 375.103,Z 537.194,A -85,B 0,C 180,E1 -12339.165,E2 -12339.165} C_VEL
LIN {X 0,Y 375.574,Z 530.219,A -85,B 0,C 180,E1 -12340.786,E2 -12340.786} C_VEL
LIN {X 0,Y 376.368,Z 521.469,A -85,B 0,C 180,E1 -12342.401,E2 -12342.401} C_VEL
LIN {X 0,Y 377.182,Z 512.491,A -85,B 0,C 180,E1 -12343.744,E2 -12343.744} C_VEL
LIN {X 0,Y 377.947,Z 501.373,A -85,B 0,C 180,E1 -12345.091,E2 -12345.091} C_VEL
LIN {X 0,Y 378.9,Z 490.114,A -85,B 0,C 180,E1 -12346.155,E2 -12346.155} C_VEL
LIN {X 0,Y 379.844,Z 477.459,A -85,B 0,C 180,E1 -12347.082,E2 -12347.082} C_VEL
LIN {X 0,Y 380.499,Z 465.142,A -85,B 0,C 180,E1 -12347.745,E2 -12347.745} C_VEL
LIN {X 0,Y 381.135,Z 451.497,A -85,B 0,C 180,E1 -12348.235,E2 -12348.235} C_VEL
LIN {X 0,Y 381.731,Z 410.479,A -85,B 0,C 180,E1 -12349.04,E2 -12349.04} C_VEL
LIN {X 0,Y 382.076,Z 371.84,A -85,B 0,C 180,E1 -12349.773,E2 -12349.773} C_VEL
LIN {X 0,Y 377.752,Z 341.923,A -85,B 0,C 180,E1 -12350.582,E2 -12350.582} C_VEL
LIN {X 0,Y 378.891,Z 327.234,A -85,B 0,C 180,E1 -12353.794,E2 -12353.794} C_VEL
LIN {X 0,Y 378.837,Z 323.527,A -85,B 0,C 180,E1 -12354.628,E2 -12354.628} C_VEL
LIN {X 0,Y 376.321,Z 310.088,A -85,B 0,C 180,E1 -12357.833,E2 -12357.833} C_VEL
LIN {X 0,Y 376.019,Z 308.647,A -85,B 0,C 180,E1 -12358.19,E2 -12358.19} C_VEL
LIN {X 0,Y 375.962,Z 308.653,A -85,B 0,C 180,E1 -12361.562,E2 -12361.562} C_VEL
LIN {X 0,Y 375.961,Z 308.65,A -85,B 0,C 180,E1 -12365.416,E2 -12365.416} C_VEL
LIN {X 0,Y 375.94,Z 308.657,A -85,B 0,C 180,E1 -12368.263,E2 -12368.263} C_VEL
LIN {X 0,Y 375.923,Z 308.655,A -85,B 0,C 180,E1 -12371.598,E2 -12371.598} C_VEL
LIN {X 0,Y 375.931,Z 308.656,A -85,B 0,C 180,E1 -12374.732,E2 -12374.732} C_VEL
LIN {X 0,Y 375.928,Z 308.659,A -85,B 0,C 180,E1 -12378.401,E2 -12378.401} C_VEL
LIN {X 0,Y 375.974,Z 308.648,A -85,B 0,C 180,E1 -12381.731,E2 -12381.731} C_VEL
LIN {X 0,Y 375.984,Z 308.648,A -85,B 0,C 180,E1 -12385.333,E2 -12385.333} C_VEL
LIN {X 0,Y 375.962,Z 308.651,A -85,B 0,C 180,E1 -12388.438,E2 -12388.438} C_VEL
LIN {X 0,Y 375.962,Z 308.649,A -85,B 0,C 180,E1 -12392.138,E2 -12392.138} C_VEL
LIN {X 0,Y 375.98,Z 308.648,A -85,B 0,C 180,E1 -12394.537,E2 -12394.537} C_VEL
LIN {X 0,Y 375.961,Z 308.65,A -85,B 0,C 180,E1 -12398.045,E2 -12398.045} C_VEL
LIN {X 0,Y 376.007,Z 308.65,A -85,B 0,C 180,E1 -12401.473,E2 -12401.473} C_VEL
LIN {X 0,Y 376.062,Z 308.637,A -85,B 0,C 180,E1 -12404.832,E2 -12404.832} C_VEL
LIN {X 0,Y 376.052,Z 308.64,A -85,B 0,C 180,E1 -12408.136,E2 -12408.136} C_VEL
LIN {X 0,Y 376.203,Z 308.625,A -85,B 0,C 180,E1 -12411.941,E2 -12411.941} C_VEL
LIN {X 0,Y 376.165,Z 308.624,A -85,B 0,C 180,E1 -12414.64,E2 -12414.64} C_VEL
LIN {X 0,Y 376.347,Z 308.606,A -85,B 0,C 180,E1 -12417.859,E2 -12417.859} C_VEL
LIN {X 0,Y 376.487,Z 308.59,A -85,B 0,C 180,E1 -12420,E2 -12420} C_VEL
LIN {X 0,Y 376.348,Z 308.608,A -85,B 0,C 180,E1 -12422.14,E2 -12422.14} C_VEL
LIN {X 0,Y 376.197,Z 308.625,A -85,B 0,C 180,E1 -12426.498,E2 -12426.498} C_VEL
LIN {X 0,Y 376.117,Z 308.63,A -85,B 0,C 180,E1 -12429.681,E2 -12429.681} C_VEL
LIN {X 0,Y 376.093,Z 308.633,A -85,B 0,C 180,E1 -12433.657,E2 -12433.657} C_VEL
LIN {X 0,Y 376.036,Z 308.641,A -85,B 0,C 180,E1 -12437.399,E2 -12437.399} C_VEL
LIN {X 0,Y 375.982,Z 308.653,A -85,B 0,C 180,E1 -12440.832,E2 -12440.832} C_VEL
LIN {X 0,Y 375.98,Z 308.647,A -85,B 0,C 180,E1 -12444.282,E2 -12444.282} C_VEL
LIN {X 0,Y 375.967,Z 308.651,A -85,B 0,C 180,E1 -12446.656,E2 -12446.656} C_VEL
LIN {X 0,Y 375.965,Z 308.649,A -85,B 0,C 180,E1 -12450.312,E2 -12450.312} C_VEL
LIN {X 0,Y 375.962,Z 308.65,A -85,B 0,C 180,E1 -12454.111,E2 -12454.111} C_VEL
LIN {X 0,Y 375.955,Z 308.65,A -85,B 0,C 180,E1 -12456.741,E2 -12456.741} C_VEL
LIN {X 0,Y 375.978,Z 308.651,A -85,B 0,C 180,E1 -12459.968,E2 -12459.968} C_VEL
LIN {X 0,Y 375.932,Z 308.66,A -85,B 0,C 180,E1 -12463.765,E2 -12463.765} C_VEL
LIN {X 0,Y 375.936,Z 308.652,A -85,B 0,C 180,E1 -12466.81,E2 -12466.81} C_VEL
LIN {X 0,Y 375.944,Z 308.653,A -85,B 0,C 180,E1 -12470.534,E2 -12470.534} C_VEL
LIN {X 0,Y 375.965,Z 308.65,A -85,B 0,C 180,E1 -12473.495,E2 -12473.495} C_VEL
LIN {X 0,Y 375.962,Z 308.652,A -85,B 0,C 180,E1 -12475.888,E2 -12475.888} C_VEL
LIN {X 0,Y 375.964,Z 308.649,A -85,B 0,C 180,E1 -12479.686,E2 -12479.686} C_VEL
LIN {X 0,Y 375.965,Z 308.649,A -85,B 0,C 180,E1 -12483.343,E2 -12483.343} C_VEL
LIN {X 0,Y 375.992,Z 308.65,A -85,B 0,C 180,E1 -12486.887,E2 -12486.887} C_VEL
LIN {X 0,Y 375.997,Z 308.647,A -85,B 0,C 180,E1 -12490.338,E2 -12490.338} C_VEL
LIN {X 0,Y 376.026,Z 308.641,A -85,B 0,C 180,E1 -12493.718,E2 -12493.718} C_VEL
LIN {X 0,Y 376.104,Z 308.639,A -85,B 0,C 180,E1 -12497.041,E2 -12497.041} C_VEL
LIN {X 0,Y 376.135,Z 308.764,A -85,B 0,C 180,E1 -12500.08,E2 -12500.08} C_VEL
LIN {X 0,Y 378.041,Z 319.372,A -85,B 0,C 180,E1 -12502.79,E2 -12502.79} C_VEL
LIN {X 0,Y 377.867,Z 322.451,A -85,B 0,C 180,E1 -12503.525,E2 -12503.525} C_VEL
LIN {X 0,Y 382.484,Z 346.789,A -85,B 0,C 180,E1 -12504.215,E2 -12504.215} C_VEL
LIN {X 0,Y 381.267,Z 429.938,A -85,B 0,C 180,E1 -12505.799,E2 -12505.799} C_VEL
LIN {X 0,Y 380.8,Z 442.834,A -85,B 0,C 180,E1 -12506.247,E2 -12506.247} C_VEL
LIN {X 0,Y 380.268,Z 455.088,A -85,B 0,C 180,E1 -12506.88,E2 -12506.88} C_VEL
LIN {X 0,Y 379.491,Z 467.256,A -85,B 0,C 180,E1 -12507.73,E2 -12507.73} C_VEL
LIN {X 0,Y 378.629,Z 478.953,A -85,B 0,C 180,E1 -12508.803,E2 -12508.803} C_VEL
LIN {X 0,Y 377.748,Z 489.355,A -85,B 0,C 180,E1 -12509.999,E2 -12509.999} C_VEL
LIN {X 0,Y 376.952,Z 498.709,A -85,B 0,C 180,E1 -12511.334,E2 -12511.334} C_VEL
LIN {X 0,Y 376.105,Z 507.755,A -85,B 0,C 180,E1 -12512.945,E2 -12512.945} C_VEL
LIN {X 0,Y 375.483,Z 515.046,A -85,B 0,C 180,E1 -12514.562,E2 -12514.562} C_VEL
LIN {X 0,Y 375.233,Z 519.96,A -85,B 0,C 180,E1 -12515.912,E2 -12515.912} C_VEL
LIN {X 0,Y 374.892,Z 524.757,A -85,B 0,C 180,E1 -12517.539,E2 -12517.539} C_VEL
LIN {X 0,Y 374.649,Z 528.436,A -85,B 0,C 180,E1 -12519.174,E2 -12519.174} C_VEL
LIN {X 0,Y 374.464,Z 531.09,A -85,B 0,C 180,E1 -12520.816,E2 -12520.816} C_VEL
LIN {X 0,Y 374.436,Z 532.853,A -85,B 0,C 180,E1 -12522.575,E2 -12522.575} C_VEL
LIN {X 0,Y 374.349,Z 533.52,A -85,B 0,C 180,E1 -12524.125,E2 -12524.125} C_VEL
LIN {X 0,Y 374.339,Z 533.505,A -85,B 0,C 180,E1 -12525.238,E2 -12525.238} C_VEL
LIN {X 0,Y 374.481,Z 532.488,A -85,B 0,C 180,E1 -12527.113,E2 -12527.113} C_VEL
LIN {X 0,Y 373.924,Z 531.665,A -85,B 0,C 180,E1 -12528.003,E2 -12528.003} C_VEL
LIN {X 0,Y 371.286,Z 529.804,A -85,B 0,C 180,E1 -12529.445,E2 -12529.445} C_VEL
LIN {X 0,Y 369.091,Z 527.905,A -85,B 0,C 180,E1 -12530.594,E2 -12530.594} C_VEL
LIN {X 0,Y 368.25,Z 526.108,A -85,B 0,C 180,E1 -12531.465,E2 -12531.465} C_VEL
LIN {X 0,Y 368.238,Z 525.407,A -85,B 0,C 180,E1 -12531.755,E2 -12531.755} C_VEL
LIN {X 0,Y 368.855,Z 520.24,A -85,B 0,C 180,E1 -12533.585,E2 -12533.585} C_VEL
LIN {X 0,Y 369.692,Z 513.897,A -85,B 0,C 180,E1 -12535.323,E2 -12535.323} C_VEL
LIN {X 0,Y 370.682,Z 506.272,A -85,B 0,C 180,E1 -12536.988,E2 -12536.988} C_VEL
LIN {X 0,Y 371.762,Z 497.546,A -85,B 0,C 180,E1 -12538.51,E2 -12538.51} C_VEL
LIN {X 0,Y 373.006,Z 487.487,A -85,B 0,C 180,E1 -12539.922,E2 -12539.922} C_VEL
LIN {X 0,Y 374.182,Z 477.064,A -85,B 0,C 180,E1 -12541.097,E2 -12541.097} C_VEL
LIN {X 0,Y 375.289,Z 465.992,A -85,B 0,C 180,E1 -12542.083,E2 -12542.083} C_VEL
LIN {X 0,Y 376.213,Z 454.47,A -85,B 0,C 180,E1 -12542.881,E2 -12542.881} C_VEL
LIN {X 0,Y 376.949,Z 441.875,A -85,B 0,C 180,E1 -12543.526,E2 -12543.526} C_VEL
LIN {X 0,Y 377.504,Z 429.221,A -85,B 0,C 180,E1 -12543.951,E2 -12543.951} C_VEL
LIN {X 0,Y 379.049,Z 348.705,A -85,B 0,C 180,E1 -12545.526,E2 -12545.526} C_VEL
LIN {X 0,Y 375.169,Z 331.42,A -85,B 0,C 180,E1 -12546.17,E2 -12546.17} C_VEL
LIN {X 0,Y 372.458,Z 324.563,A -85,B 0,C 180,E1 -12546.52,E2 -12546.52} C_VEL
LIN {X 0,Y 371.789,Z 322.675,A -85,B 0,C 180,E1 -12546.632,E2 -12546.632} C_VEL
LIN {X 0,Y 369.776,Z 313.129,A -85,B 0,C 180,E1 -12549.241,E2 -12549.241} C_VEL
LIN {X 0,Y 368.877,Z 309.539,A -85,B 0,C 180,E1 -12550.292,E2 -12550.292} C_VEL
LIN {X 0,Y 368.875,Z 309.537,A -85,B 0,C 180,E1 -12553.615,E2 -12553.615} C_VEL
LIN {X 0,Y 368.877,Z 309.531,A -85,B 0,C 180,E1 -12556.695,E2 -12556.695} C_VEL
LIN {X 0,Y 368.876,Z 309.535,A -85,B 0,C 180,E1 -12559.647,E2 -12559.647} C_VEL
LIN {X 0,Y 368.891,Z 309.536,A -85,B 0,C 180,E1 -12563.144,E2 -12563.144} C_VEL
LIN {X 0,Y 368.887,Z 309.516,A -85,B 0,C 180,E1 -12566.461,E2 -12566.461} C_VEL
LIN {X 0,Y 368.904,Z 309.533,A -85,B 0,C 180,E1 -12569.044,E2 -12569.044} C_VEL
LIN {X 0,Y 368.907,Z 309.531,A -85,B 0,C 180,E1 -12571.558,E2 -12571.558} C_VEL
LIN {X 0,Y 368.889,Z 309.531,A -85,B 0,C 180,E1 -12575.22,E2 -12575.22} C_VEL
LIN {X 0,Y 368.911,Z 309.527,A -85,B 0,C 180,E1 -12577.604,E2 -12577.604} C_VEL
LIN {X 0,Y 368.912,Z 309.528,A -85,B 0,C 180,E1 -12581.104,E2 -12581.104} C_VEL
LIN {X 0,Y 368.93,Z 309.527,A -85,B 0,C 180,E1 -12584.533,E2 -12584.533} C_VEL
LIN {X 0,Y 369.048,Z 309.504,A -85,B 0,C 180,E1 -12586.79,E2 -12586.79} C_VEL
LIN {X 0,Y 369.048,Z 309.511,A -85,B 0,C 180,E1 -12590.131,E2 -12590.131} C_VEL
LIN {X 0,Y 369.142,Z 309.498,A -85,B 0,C 180,E1 -12593.441,E2 -12593.441} C_VEL
LIN {X 0,Y 369.284,Z 309.476,A -85,B 0,C 180,E1 -12597.819,E2 -12597.819} C_VEL
LIN {X 0,Y 369.285,Z 309.475,A -85,B 0,C 180,E1 -12602.182,E2 -12602.182} C_VEL
LIN {X 0,Y 369.169,Z 309.494,A -85,B 0,C 180,E1 -12606.559,E2 -12606.559} C_VEL
LIN {X 0,Y 369.051,Z 309.509,A -85,B 0,C 180,E1 -12609.869,E2 -12609.869} C_VEL
LIN {X 0,Y 369.029,Z 309.505,A -85,B 0,C 180,E1 -12613.773,E2 -12613.773} C_VEL
LIN {X 0,Y 368.983,Z 309.509,A -85,B 0,C 180,E1 -12617.743,E2 -12617.743} C_VEL
LIN {X 0,Y 368.902,Z 309.531,A -85,B 0,C 180,E1 -12621.222,E2 -12621.222} C_VEL
LIN {X 0,Y 368.903,Z 309.527,A -85,B 0,C 180,E1 -12623.875,E2 -12623.875} C_VEL
LIN {X 0,Y 368.864,Z 309.532,A -85,B 0,C 180,E1 -12627.212,E2 -12627.212} C_VEL
LIN {X 0,Y 368.923,Z 309.529,A -85,B 0,C 180,E1 -12630.954,E2 -12630.954} C_VEL
LIN {X 0,Y 368.923,Z 309.528,A -85,B 0,C 180,E1 -12635.002,E2 -12635.002} C_VEL
LIN {X 0,Y 368.871,Z 309.531,A -85,B 0,C 180,E1 -12638.635,E2 -12638.635} C_VEL
LIN {X 0,Y 368.866,Z 309.529,A -85,B 0,C 180,E1 -12642.009,E2 -12642.009} C_VEL
LIN {X 0,Y 368.875,Z 309.534,A -85,B 0,C 180,E1 -12645.177,E2 -12645.177} C_VEL
LIN {X 0,Y 368.877,Z 309.542,A -85,B 0,C 180,E1 -12648.179,E2 -12648.179} C_VEL
LIN {X 0,Y 368.901,Z 309.535,A -85,B 0,C 180,E1 -12651.362,E2 -12651.362} C_VEL
LIN {X 0,Y 368.934,Z 309.523,A -85,B 0,C 180,E1 -12655.148,E2 -12655.148} C_VEL
LIN {X 0,Y 368.927,Z 309.533,A -85,B 0,C 180,E1 -12659.048,E2 -12659.048} C_VEL
LIN {X 0,Y 368.946,Z 309.653,A -85,B 0,C 180,E1 -12659.486,E2 -12659.486} C_VEL
LIN {X 0,Y 371.428,Z 320.101,A -85,B 0,C 180,E1 -12662.328,E2 -12662.328} C_VEL
LIN {X 0,Y 373.143,Z 329.301,A -85,B 0,C 180,E1 -12664.698,E2 -12664.698} C_VEL
LIN {X 0,Y 373.322,Z 332.763,A -85,B 0,C 180,E1 -12665.535,E2 -12665.535} C_VEL
LIN {X 0,Y 372.369,Z 341.342,A -85,B 0,C 180,E1 -12667.486,E2 -12667.486} C_VEL
LIN {X 0,Y 376.679,Z 362.453,A -85,B 0,C 180,E1 -12668.251,E2 -12668.251} C_VEL
LIN {X 0,Y 378.647,Z 374.51,A -85,B 0,C 180,E1 -12668.64,E2 -12668.64} C_VEL
LIN {X 0,Y 377.276,Z 449.824,A -85,B 0,C 180,E1 -12670.126,E2 -12670.126} C_VEL
LIN {X 0,Y 376.54,Z 462.949,A -85,B 0,C 180,E1 -12670.583,E2 -12670.583} C_VEL
LIN {X 0,Y 375.613,Z 475.585,A -85,B 0,C 180,E1 -12671.242,E2 -12671.242} C_VEL
LIN {X 0,Y 374.464,Z 487.655,A -85,B 0,C 180,E1 -12672.103,E2 -12672.103} C_VEL
LIN {X 0,Y 373.238,Z 499.136,A -85,B 0,C 180,E1 -12673.173,E2 -12673.173} C_VEL
LIN {X 0,Y 371.947,Z 509.5,A -85,B 0,C 180,E1 -12674.381,E2 -12674.381} C_VEL
LIN {X 0,Y 370.919,Z 518.846,A -85,B 0,C 180,E1 -12675.741,E2 -12675.741} C_VEL
LIN {X 0,Y 369.751,Z 527.89,A -85,B 0,C 180,E1 -12677.375,E2 -12677.375} C_VEL
LIN {X 0,Y 368.894,Z 535.199,A -85,B 0,C 180,E1 -12679.018,E2 -12679.018} C_VEL
LIN {X 0,Y 368.232,Z 541.079,A -85,B 0,C 180,E1 -12680.665,E2 -12680.665} C_VEL
LIN {X 0,Y 367.795,Z 545.731,A -85,B 0,C 180,E1 -12682.314,E2 -12682.314} C_VEL
LIN {X 0,Y 367.515,Z 549.234,A -85,B 0,C 180,E1 -12683.935,E2 -12683.935} C_VEL
LIN {X 0,Y 367.437,Z 551.856,A -85,B 0,C 180,E1 -12685.613,E2 -12685.613} C_VEL
LIN {X 0,Y 367.377,Z 553.069,A -85,B 0,C 180,E1 -12686.711,E2 -12686.711} C_VEL
LIN {X 0,Y 367.403,Z 554.226,A -85,B 0,C 180,E1 -12688.905,E2 -12688.905} C_VEL
LIN {X 0,Y 367.457,Z 554.223,A -85,B 0,C 180,E1 -12690.001,E2 -12690.001} C_VEL
LIN {X 0,Y 367.42,Z 553.831,A -85,B 0,C 180,E1 -12691.097,E2 -12691.097} C_VEL
LIN {X 0,Y 367.376,Z 553.009,A -85,B 0,C 180,E1 -12692.194,E2 -12692.194} C_VEL
LIN {X 0,Y 367.382,Z 551.77,A -85,B 0,C 180,E1 -12693.291,E2 -12693.291} C_VEL
LIN {X 0,Y 367.469,Z 549.132,A -85,B 0,C 180,E1 -12694.938,E2 -12694.938} C_VEL
LIN {X 0,Y 367.565,Z 545.459,A -85,B 0,C 180,E1 -12696.589,E2 -12696.589} C_VEL
LIN {X 0,Y 367.807,Z 540.656,A -85,B 0,C 180,E1 -12698.24,E2 -12698.24} C_VEL
LIN {X 0,Y 368.318,Z 533.447,A -85,B 0,C 180,E1 -12700.167,E2 -12700.167} C_VEL
LIN {X 0,Y 368.961,Z 525.554,A -85,B 0,C 180,E1 -12701.817,E2 -12701.817} C_VEL
LIN {X 0,Y 369.647,Z 517.484,A -85,B 0,C 180,E1 -12703.189,E2 -12703.189} C_VEL
LIN {X 0,Y 370.537,Z 507.866,A -85,B 0,C 180,E1 -12704.526,E2 -12704.526} C_VEL
LIN {X 0,Y 371.385,Z 496.621,A -85,B 0,C 180,E1 -12705.786,E2 -12705.786} C_VEL
LIN {X 0,Y 372.278,Z 485.83,A -85,B 0,C 180,E1 -12706.733,E2 -12706.733} C_VEL
LIN {X 0,Y 373.188,Z 472.818,A -85,B 0,C 180,E1 -12707.608,E2 -12707.608} C_VEL
LIN {X 0,Y 373.897,Z 460.376,A -85,B 0,C 180,E1 -12708.21,E2 -12708.21} C_VEL
LIN {X 0,Y 374.37,Z 447.463,A -85,B 0,C 180,E1 -12708.612,E2 -12708.612} C_VEL
LIN {X 0,Y 375.401,Z 373.495,A -85,B 0,C 180,E1 -12710.036,E2 -12710.036} C_VEL
LIN {X 0,Y 370.811,Z 341.791,A -85,B 0,C 180,E1 -12710.9,E2 -12710.9} C_VEL
LIN {X 0,Y 371.925,Z 327.996,A -85,B 0,C 180,E1 -12713.972,E2 -12713.972} C_VEL
LIN {X 0,Y 371.779,Z 324.17,A -85,B 0,C 180,E1 -12714.854,E2 -12714.854} C_VEL
LIN {X 0,Y 369.52,Z 312.158,A -85,B 0,C 180,E1 -12717.774,E2 -12717.774} C_VEL
LIN {X 0,Y 368.968,Z 309.524,A -85,B 0,C 180,E1 -12718.438,E2 -12718.438} C_VEL
LIN {X 0,Y 368.903,Z 309.532,A -85,B 0,C 180,E1 -12722.238,E2 -12722.238} C_VEL
LIN {X 0,Y 368.933,Z 309.525,A -85,B 0,C 180,E1 -12725.002,E2 -12725.002} C_VEL
LIN {X 0,Y 368.881,Z 309.533,A -85,B 0,C 180,E1 -12728.634,E2 -12728.634} C_VEL
LIN {X 0,Y 368.875,Z 309.536,A -85,B 0,C 180,E1 -12732.008,E2 -12732.008} C_VEL
LIN {X 0,Y 368.884,Z 309.531,A -85,B 0,C 180,E1 -12735.176,E2 -12735.176} C_VEL
LIN {X 0,Y 368.879,Z 309.535,A -85,B 0,C 180,E1 -12738.177,E2 -12738.177} C_VEL
LIN {X 0,Y 368.907,Z 309.528,A -85,B 0,C 180,E1 -12741.361,E2 -12741.361} C_VEL
LIN {X 0,Y 368.941,Z 309.527,A -85,B 0,C 180,E1 -12745.147,E2 -12745.147} C_VEL
LIN {X 0,Y 368.934,Z 309.53,A -85,B 0,C 180,E1 -12749.047,E2 -12749.047} C_VEL
LIN {X 0,Y 368.903,Z 309.532,A -85,B 0,C 180,E1 -12752.791,E2 -12752.791} C_VEL
LIN {X 0,Y 368.932,Z 309.525,A -85,B 0,C 180,E1 -12756.119,E2 -12756.119} C_VEL
LIN {X 0,Y 368.94,Z 309.525,A -85,B 0,C 180,E1 -12759.947,E2 -12759.947} C_VEL
LIN {X 0,Y 368.973,Z 309.526,A -85,B 0,C 180,E1 -12763.398,E2 -12763.398} C_VEL
LIN {X 0,Y 369.062,Z 309.509,A -85,B 0,C 180,E1 -12766.79,E2 -12766.79} C_VEL
LIN {X 0,Y 369.067,Z 309.511,A -85,B 0,C 180,E1 -12770.131,E2 -12770.131} C_VEL
LIN {X 0,Y 369.189,Z 309.495,A -85,B 0,C 180,E1 -12773.441,E2 -12773.441} C_VEL
LIN {X 0,Y 369.311,Z 309.482,A -85,B 0,C 180,E1 -12777.819,E2 -12777.819} C_VEL
LIN {X 0,Y 369.456,Z 309.465,A -85,B 0,C 180,E1 -12780,E2 -12780} C_VEL
LIN {X 0,Y 369.312,Z 309.485,A -85,B 0,C 180,E1 -12782.181,E2 -12782.181} C_VEL
LIN {X 0,Y 369.164,Z 309.501,A -85,B 0,C 180,E1 -12786.559,E2 -12786.559} C_VEL
LIN {X 0,Y 369.067,Z 309.509,A -85,B 0,C 180,E1 -12789.868,E2 -12789.868} C_VEL
LIN {X 0,Y 369.041,Z 309.511,A -85,B 0,C 180,E1 -12793.772,E2 -12793.772} C_VEL
LIN {X 0,Y 368.994,Z 309.517,A -85,B 0,C 180,E1 -12797.742,E2 -12797.742} C_VEL
LIN {X 0,Y 368.913,Z 309.531,A -85,B 0,C 180,E1 -12801.22,E2 -12801.22} C_VEL
LIN {X 0,Y 368.941,Z 309.528,A -85,B 0,C 180,E1 -12804.776,E2 -12804.776} C_VEL
LIN {X 0,Y 368.933,Z 309.525,A -85,B 0,C 180,E1 -12808.44,E2 -12808.44} C_VEL
LIN {X 0,Y 368.913,Z 309.531,A -85,B 0,C 180,E1 -12810.987,E2 -12810.987} C_VEL
LIN {X 0,Y 368.939,Z 309.525,A -85,B 0,C 180,E1 -12814.853,E2 -12814.853} C_VEL
LIN {X 0,Y 368.905,Z 309.528,A -85,B 0,C 180,E1 -12818.638,E2 -12818.638} C_VEL
LIN {X 0,Y 368.877,Z 309.536,A -85,B 0,C 180,E1 -12822.008,E2 -12822.008} C_VEL
LIN {X 0,Y 368.881,Z 309.532,A -85,B 0,C 180,E1 -12825.175,E2 -12825.175} C_VEL
LIN {X 0,Y 368.876,Z 309.536,A -85,B 0,C 180,E1 -12828.176,E2 -12828.176} C_VEL
LIN {X 0,Y 368.882,Z 309.532,A -85,B 0,C 180,E1 -12831.365,E2 -12831.365} C_VEL
LIN {X 0,Y 368.938,Z 309.524,A -85,B 0,C 180,E1 -12835.146,E2 -12835.146} C_VEL
LIN {X 0,Y 368.931,Z 309.526,A -85,B 0,C 180,E1 -12839.046,E2 -12839.046} C_VEL
LIN {X 0,Y 368.9,Z 309.533,A -85,B 0,C 180,E1 -12842.791,E2 -12842.791} C_VEL
LIN {X 0,Y 368.94,Z 309.525,A -85,B 0,C 180,E1 -12846.114,E2 -12846.114} C_VEL
LIN {X 0,Y 368.937,Z 309.524,A -85,B 0,C 180,E1 -12849.946,E2 -12849.946} C_VEL
LIN {X 0,Y 368.969,Z 309.522,A -85,B 0,C 180,E1 -12853.398,E2 -12853.398} C_VEL
LIN {X 0,Y 369.058,Z 309.513,A -85,B 0,C 180,E1 -12856.789,E2 -12856.789} C_VEL
LIN {X 0,Y 369.074,Z 309.655,A -85,B 0,C 180,E1 -12859.854,E2 -12859.854} C_VEL
LIN {X 0,Y 371.044,Z 320.401,A -85,B 0,C 180,E1 -12862.654,E2 -12862.654} C_VEL
LIN {X 0,Y 370.919,Z 322.746,A -85,B 0,C 180,E1 -12863.198,E2 -12863.198} C_VEL
LIN {X 0,Y 375.729,Z 347.906,A -85,B 0,C 180,E1 -12863.928,E2 -12863.928} C_VEL
LIN {X 0,Y 374.421,Z 429.862,A -85,B 0,C 180,E1 -12865.512,E2 -12865.512} C_VEL
LIN {X 0,Y 373.957,Z 442.51,A -85,B 0,C 180,E1 -12865.954,E2 -12865.954} C_VEL
